// ── UPPER ─────────────────────────────────────────────────────────────────────
rawTorqueUpper := upperMasterTorqueFeedback;
instsFT_PT1UpperTorqueFilter( in := rawTorqueUpper, 
							   T := torqueFilterTime, 
							   K := 1.0, 
							   out => filteredTorqueUpper );
							   

// Master cap and base limit (never exceed master)
capMasterUpper := LIMIT(torqueLimitMinPct, filteredTorqueUpper, torqueLimitMaxPct);
baseLimitUpper := MIN(
    capMasterUpper,
    LIMIT(torqueLimitMinPct, filteredTorqueUpper + slaveTorqueOfsset, torqueLimitMaxPct)
);

IF NOT enableTorquePid THEN
    upperSlave1DriveTorqueRefPct := capMasterUpper;
    upperSlave2DriveTorqueRefPct := capMasterUpper;
ELSE
    directTorqueUpper := LIMIT(torqueLimitMinPct, baseLimitUpper - torqueTrimLimit, capMasterUpper);
    avgTorqueUpper    := 0.5 * (upperSlave1TorqueFeedback + upperSlave2TorqueFeedback);

    instCTRL_PID_UpperTorqueTrim(
        ACT := avgTorqueUpper,
        SET := baseLimitUpper,
        MAN := NOT enableTorquePid,   // manual when disabled (tracks 0)
        M_I := 0.0,
        RST := FALSE,
        KP  := torqueCtrlKp,
        TN  := torqueCtrlTn,
        TV  := torqueCtrlTv,
        LL  := 0.0,                   // unipolar: only add
        LH  := torqueTrimLimit,
        Y   => trimUp
    );

    upperSlave1DriveTorqueRefPct := LIMIT(torqueLimitMinPct, directTorqueUpper + trimUp, capMasterUpper);
    upperSlave2DriveTorqueRefPct := LIMIT(torqueLimitMinPct, directTorqueUpper + trimUp, capMasterUpper);
END_IF;


// ── LOWER ─────────────────────────────────────────────────────────────────────
rawTorqueLower := lowerMasterTorqueFeedback;
instsFT_PT1LowerTorqueFilter( in := rawTorqueLower, T := torqueFilterTime, K := 1.0, out => filteredTorqueLower );

capMasterLower := LIMIT(torqueLimitMinPct, filteredTorqueLower, torqueLimitMaxPct);
baseLimitLower := MIN(
    capMasterLower,
    LIMIT(torqueLimitMinPct, filteredTorqueLower + slaveTorqueOfsset, torqueLimitMaxPct)
);

IF NOT enableTorquePid THEN
    lowerSlave1DriveTorqueRefPct := capMasterLower;
    lowerSlave2DriveTorqueRefPct := capMasterLower;
ELSE
    directTorqueLower := LIMIT(torqueLimitMinPct, baseLimitLower - torqueTrimLimit, capMasterLower);
    avgTorqueLower    := 0.5 * (lowerSlave1TorqueFeedback + lowerSlave2TorqueFeedback);

    instCTRL_PID_LowerTorqueTrim(
        ACT := avgTorqueLower,
        SET := baseLimitLower,
        MAN := NOT enableTorquePid,
        M_I := 0.0,
        RST := FALSE,
        KP  := torqueCtrlKp,
        TN  := torqueCtrlTn,
        TV  := torqueCtrlTv,
        LL  := 0.0,
        LH  := torqueTrimLimit,
        Y   => trimLo
    );

    lowerSlave1DriveTorqueRefPct := LIMIT(torqueLimitMinPct, directTorqueLower + trimLo, capMasterLower);
    lowerSlave2DriveTorqueRefPct := LIMIT(torqueLimitMinPct, directTorqueLower + trimLo, capMasterLower);
END_IF;
END_METHOD

END_FUNCTION_BLOCK

// ---- Function Blocks/PaperMachine/Auxiliary/FB_Gen_SRamp.TcPOU
FUNCTION_BLOCK FB_Gen_SRamp
VAR_INPUT
	X : REAL;
	A_UP : REAL  := 1.0;
	A_DN :REAL  := -1.0;;
	VU_MAX : REAL := 1.0;
	VD_MAX : REAL := -1.0;
	LIMIT_HIGH : REAL := 100.0;
	LIMIT_LOW : REAL := -100.0;
	RST : BOOL;
END_VAR
VAR_OUTPUT
	Y : REAL;
	V : REAL;
END_VAR
VAR
	cycle_time : TC_S;
	init: BOOL;
END_VAR

(* read the system_time in microseconds *)
cycle_time();

(* assure range of inputs *)
A_up := MAX(0.0, A_UP);
A_dn := MIN(0.0, A_dn);
VU_max := MAX(0.0, VU_max);
VD_max := MIN(0.0, VD_MAX);

(* calculate the output offset *)
IF rst OR NOT init THEN
	init := TRUE;
	Y := 0.0;
	V := 0.0;
ELSIF X = Y THEN
	v := 0.0;
ELSIF X > Y THEN
	(* output is too low >> ramp up and brake at the end *)
	(* accelerate the speed and limit to vu_max *)
	v := MIN(v + A_UP * cycle_time.TC, vu_max);
	(* calculate the max speed to be able to brake and select the lowest *)
	v := MIN(SQRT((Y-X) * 2.0 * A_DN), v);
	(* calculate the output and obey limits *)
	y := LIMIT(limit_low, y + MIN(v * cycle_time.TC, X-Y), limit_high);
ELSIF X < Y THEN
	(* output is too high >> ramp dn and brake at the end *)
	(* accelerate the speed and limit to vd_max *)
	v := MAX(v + A_DN * cycle_time.TC, vd_max);
	(* calculate the max speed to be able to brake and select the lowest *)
	v := MAX(-SQRT((Y-X) * 2.0 * A_UP), v);
	(* calculate the output and obey limits *)
	y := LIMIT(limit_low, y + MAX(v * cycle_time.TC, X-Y), limit_high);
END_IF;


(* revision history
hm	13. mar. 2008	rev 1.0
	original version

hm	11. mar. 2009	rev 1.1
	real constants updated to new systax using dot																																																																																																																																																																																																																																																																																																																																																																																																																																																																																																																																																																																																																																																																																																																																																																																																																																																																																																																																																																																																																																																											

*)

END_FUNCTION_BLOCK

// ---- Function Blocks/PaperMachine/DriveControl/FB_PressSectionDriveControl_V2.TcPOU
FUNCTION_BLOCK FB_PressSectionDriveControl_V2

VAR_INPUT

    //────────────────────────────────────────────
    // GROUP / INTERLOCKS
    //────────────────────────────────────────────
    startGroup              : BOOL; // Start command (pulse) / Comando de partida (pulso)
    stopGroup               : BOOL; // Stop command (level) / Comando de parada (nível)
    groupReset              : BOOL; // Fault reset / Reset de falhas do grupo
    groupFastStop           : BOOL;  // EN: Reset group faults / PT: Reset de falhas do grupo
	
    //────────────────────────────────────────────
    // AUXILIARY MOTORS — INDICATORS & COMMANDS
    //────────────────────────────────────────────
    grouSpeedDifIncCmd         : BOOL; // Lamp: offset increasing / Lâmpada: aumento de offset
    grouSpeedDifDecCmd         : BOOL; // Lamp: offset decreasing / Lâmpada: redução de offset
	
    //────────────────────────────────────────────
    // SPEED ADJUSTMENTS / OFFSET TUNING
    //────────────────────────────────────────────
    groupRecoverSpeedCmd    : BOOL; // Recover speed while TRUE / Recuperar velocidade enquanto TRUE


    //────────────────────────────────────────────
    // DRIVE STATUS INPUTS — PRESS SECTION (2 MOTORS)
    //────────────────────────────────────────────
    firstPressReady         : BOOL; // First press (MASTER) ready / Prensa 1 (mestre) pronto
    secondPressReady        : BOOL; // Second press (SLAVE) ready / Prensa 2 (escravo) pronto
	paperPresenceSensor : BOOL;

    //────────────────────────────────────────────
    // SPEED SETPOINTS / MODE
    //────────────────────────────────────────────
    groupAutoSpeedMPM       : REAL; // Auto mode speed [m/min] / Velocidade em modo automático [m/min]
    groupManualSpeedMPM     : REAL := 50.0; // Manual mode speed / Velocidade em modo manual
    groupSpeedAutoMan       : BOOL; // Speed mode: 0=Manual, 1=Auto / Modo de velocidade: 0=Manual, 1=Automático

    //────────────────────────────────────────────
    // SPEED & TORQUE FEEDBACKS
    //────────────────────────────────────────────
    firstPressSpeedFeedback : REAL; // First press speed feedback / Velocidade medida da prensa 1
    firstPressTorqueFeedback: REAL; // First press torque feedback / Torque da prensa 1
    secondPressSpeedFeedback: REAL; // Second press speed feedback / Velocidade medida da prensa 2
    secondPressTorqueFeedback: REAL; // Second press torque feedback / Torque da prensa 2


    //──── Upper Felt 1 Stretcher ────
    upperFelt1StretcherCmdFwd     : BOOL; // Run forward / Comando para frente
    upperFelt1StretcherCmdRev     : BOOL; // Run reverse / Comando para trás
    upperFelt1StretcherFault      : BOOL; // Fault detected / Falha detectada
    upperFelt1StretcherLimitFwd   : BOOL; // End limit forward / Fim de curso frente
    upperFelt1StretcherLimitRev   : BOOL; // End limit reverse / Fim de curso trás

    //──── Upper Felt 2 Stretcher ────
    upperFelt2StretcherCmdFwd     : BOOL; // Run forward / Comando para frente
    upperFeltt2tretcherCmdRev     : BOOL; // Run reverse / Comando para trás (corrigir nome!)
    upperFeltS2tretcherFault      : BOOL; // Fault detected / Falha detectada
    upperFeltS2tretcherLimitFwd   : BOOL; // End limit forward / Fim de curso frente
    upperFeltS2tretcherLimitRev   : BOOL; // End limit reverse / Fim de curso trás

    //──── Lower Felt Stretcher ────
    lowerFeltStretcherCmdFwd      : BOOL;
    lowerFeltStretcherCmdRev      : BOOL;
    lowerFeltStretcherFault       : BOOL;
    lowerFeltStretcherLimitFwd    : BOOL;
    lowerFeltStretcherLimitRev    : BOOL;

    //──── Upper Infeed Roll ────
    upperInfeedRollCmdFwd         : BOOL;
    upperInfeedRollCmdRev         : BOOL;
    upperInfeedRollFault          : BOOL;
    upperInfeedRollLimitFwd       : BOOL;
    upperInfeedRollLimitRev       : BOOL;

    //──── Lower Infeed Roll ────
    lowerInfeedRollCmdFwd         : BOOL;
    lowerInfeedRollCmdRev         : BOOL;
    lowerInfeedRollFault          : BOOL;
    lowerInfeedRollLimitFwd       : BOOL;
    lowerInfeedRollLimitRev       : BOOL;

    //────────────────────────────────────────────
    // FELT EDGE / RUNNING SAFETY SENSORS
    //────────────────────────────────────────────
    pressSectionUpperFelt1OverrunSensorOperatorSide : BOOL; // Operator side / Lado operador
    pressSectionUpperFelt1OverrunSensorDriveSide    : BOOL; // Drive side / Lado comando

    pressSectionUpperFelt2OverrunSensorOperatorSide : BOOL;
    pressSectionUpperFelt2OverrunSensorDriveSide    : BOOL;

    pressSectionLowerFeltOverrunSensorOperatorSide  : BOOL;
    pressSectionLowerFeltOverrunSensorDriveSide     : BOOL;

	
	machineConfig			:  PaperMachine_TypeHmiConfig;
	
END_VAR



VAR_OUTPUT

    //────────────────────────────────────────────
    // STATE / DIAGNOSTICS
    //────────────────────────────────────────────
    deviceState                 : STRING; // Current state string / Estado atual em texto
    statusCode                  : INT;    // 0=Idle, 1=Starting, 2=Running, 3=Fault
    groupFault                  : BOOL;   // TRUE if any group fault active / Falha geral do grupo
	speedDif						: REAL;

    //────────────────────────────────────────────
    // SPEED REFERENCES (TO DRIVES) AND DISPLAY
    //────────────────────────────────────────────
    firstPressSpeedSetpointRPM  		: REAL; // Master speed reference [%] / Referência de velocidade mestre
    secondPressSpeedSetpointRPM 		: REAL; // Slave speed reference [%] / Referência de velocidade escravo 
	
	firstPressSpeedFeedbackRPM  		: REAL; // Master speed reference [%] / Referência de velocidade mestre
    secondPressSpeedFeedbackRPM 		: REAL; // Slave speed reference [%] / Referência de velocidade escravo 
	
	firstPressSpeedFeedbackMPM  		: REAL; // Master speed reference [%] / Referência de velocidade mestre
    secondPressSpeedFeedbackMPM 		: REAL; // Slave speed reference [%] / Referência de velocidade escravo 

	firstPressTorqueFeedbackPct  		: REAL; // Master speed reference [%] / Referência de velocidade mestre
    secondPressTorqueFeedbackPct 		: REAL; // Slave speed reference [%] / Referência de velocidade escravo 
	
	
	nextGroupSpeedRefMPM        : REAL; // Next group speed [m/min] / Velocidade do próximo grupo [m/min]

    //────────────────────────────────────────────
    // TORQUE REFERENCES / LIMITS (SLAVE)
    //────────────────────────────────────────────
    firstPressTorqueRefPct : REAL; // Torque setpoint for slave / Referência de torque escravo
//    secondPressTorqueRefPct : REAL; // Torque setpoint for slave / Referência de torque escravo

    //────────────────────────────────────────────
    // DRIVE COMMANDS (ENABLE / RESET)
    //────────────────────────────────────────────
    firstPressDriveEnable        : BOOL; // Enable master drive / Habilita drive mestre
    firstPressDriveReset         : BOOL; // Reset master drive fault / Reset falha drive mestre
    secondPressDriveEnable       : BOOL; // Enable slave drive / Habilita drive escravo
    secondPressDriveReset        : BOOL; // Reset slave drive fault / Reset falha drive escravo

    //────────────────────────────────────────────
    // STATUS CODES (PER DRIVE)
    //────────────────────────────────────────────
    firstPressStatusCode        : INT; // 0=Idle, 1=Start, 2=Run, 3=Fault / Código de status da prensa 1
    secondPressStatusCode       : INT; // Código de status da prensa 2

    //────────────────────────────────────────────
    // AUXILIARY MOTORS — DIRECT START OUTPUTS
    //────────────────────────────────────────────
    upperFelt1StretcherRunFwd   : BOOL; // Run forward / Rodar para frente
    upperFelt1StretcherRunRev   : BOOL; // Run reverse / Rodar para trás

    upperFelt2StretcherRunFwd   : BOOL;
    upperFelt2StretcherRunRev   : BOOL;

    lowerFeltStretcherRunFwd    : BOOL;
    lowerFeltStretcherRunRev    : BOOL;

    upperInfeedRollRunFwd       : BOOL;
    upperInfeedRollRunRev       : BOOL;

    lowerInfeedRollRunFwd       : BOOL;
    lowerInfeedRollRunRev       : BOOL;

    //────────────────────────────────────────────
    // HMI ALARMS STRUCTURE
    //────────────────────────────────────────────
    hmiAlarms                   : PaperMachine_TypeHmiAlarms; // Alarm structure / Estrutura de alarmes

END_VAR




VAR
 
	instFB_GroupDriveControl_V1 : FB_GroupDriveControl_V1;
	instFB_GroupSpeedControl_V1 : FB_GroupSpeedControl_V1;
	instFB_GroupDisplayFilters_V1 : FB_GroupDisplayFilters_V1;
	instFB_GroupTorqueTrimControl_V1 : FB_GroupTorqueTrimControl_V1;

	instFB_GroupTorqueTrimControl_V2: FB_GroupTorqueTrimControl_V2;
	speedDifError: BOOL;
	speedDifCheck: REAL;
	instTONFeltOverrunDelay: TON;
	instTOF_PaperPresenseDelay: TOF;	
	
END_VAR

VAR PERSISTENT

END_VAR

// ─────────────────────────────────────────────────────────────────────────────
// MAIN CALL SEQUENCE
// ─────────────────────────────────────────────────────────────────────────────

_GroupControl();          // 1) State machine: edges, enables, stop modes
_StateDisplay();
_SpeedDifferenceCheck();  // 4) Speed difference monitor & trip
_auxiliaryControls();

_alarmsDisplay();

METHOD _alarmsDisplay
VAR_INPUT
END_VAR
(*
//==============================================================
// FAULT EVALUATION — PER CONDITION (flags only; no global set)
//==============================================================

//----------------------------
// PRESS SECTION DRIVES
//----------------------------
hmiAlarms.pressSectionFirstPressFaultAlarm  := firstPressVfdFaultFeedback;
hmiAlarms.pressSectionSecondPressFaultAlarm := secondPressVfdFaultFeedback;

//----------------------------
// PRESS SECTION AUXILIARIES
//----------------------------
hmiAlarms.pressSectionUpperFeltStretcherFaultAlarm := upperFelt1StretcherFault;
hmiAlarms.pressSectionLowerFeltStretcherFaultAlarm := lowerFeltStretcherFault;
hmiAlarms.pressSectionUpperInfeedRollFaultAlarm    := upperInfeedRollFault;
hmiAlarms.pressSectionLowerInfeedRollFaultAlarm    := lowerInfeedRollFault;


//==============================================================
// PRESS SECTION — FELT EDGE OVERRUN ALARMS (DIRECT SENSORS)
//==============================================================

hmiAlarms.pressSectionUpperFelt1OverrunOperatorSideAlarm := pressSectionUpperFelt1OverrunSensorOperatorSide;
hmiAlarms.pressSectionUpperFelt1OverrunDriveSideAlarm    := pressSectionUpperFelt1OverrunSensorDriveSide;

hmiAlarms.pressSectionUpperFelt2OverrunOperatorSideAlarm := pressSectionUpperFelt2OverrunSensorOperatorSide;
hmiAlarms.pressSectionUpperFelt2OverrunDriveSideAlarm    := pressSectionUpperFelt2OverrunSensorDriveSide;

hmiAlarms.pressSectionLowerFeltOverrunOperatorSideAlarm := pressSectionLowerFeltOverrunSensorOperatorSide;
hmiAlarms.pressSectionLowerFeltOverrunDriveSideAlarm    := pressSectionLowerFeltOverrunSensorDriveSide;


//----------------------------
// PRESS SECTION GROUP FAULT STATUS
//----------------------------
groupFault :=
    hmiAlarms.pressSectionFirstPressFaultAlarm 
	OR hmiAlarms.pressSectionSecondPressFaultAlarm 
	OR hmiAlarms.pressFelt1OverrunOperatorSideAlarm
	OR hmiAlarms.pressFelt1OverrunDriveSideAlarm
	OR hmiAlarms.pressFelt2OverrunOperatorSideAlarm
	OR hmiAlarms.pressFelt2OverrunDriveSideAlarm
	OR hmiAlarms.pressFelt3OverrunOperatorSideAlarm
	OR hmiAlarms.pressFelt3OverrunDriveSideAlarm;


*)
//==============================================================
// FAULT EVALUATION — PER CONDITION (flags only; no global set)
//==============================================================

//----------------------------
// PRESS SECTION DRIVES
//----------------------------
//hmiAlarms.pressSectionFirstPressFaultAlarm  := firstPressVfdFaultFeedback;
//hmiAlarms.pressSectionSecondPressFaultAlarm := secondPressVfdFaultFeedback;

//----------------------------
// PRESS SECTION AUXILIARIES
//----------------------------
hmiAlarms.pressSectionUpperFeltStretcherFaultAlarm := upperFelt1StretcherFault;
hmiAlarms.pressSectionLowerFeltStretcherFaultAlarm := lowerFeltStretcherFault;
hmiAlarms.pressSectionUpperInfeedRollFaultAlarm    := upperInfeedRollFault;
hmiAlarms.pressSectionLowerInfeedRollFaultAlarm    := lowerInfeedRollFault;


//==============================================================
// PRESS SECTION — FELT EDGE OVERRUN ALARMS (DIRECT SENSORS)
//==============================================================

hmiAlarms.pressSectionUpperFelt1OverrunOperatorSideAlarm := pressSectionUpperFelt1OverrunSensorOperatorSide;
hmiAlarms.pressSectionUpperFelt1OverrunDriveSideAlarm    := pressSectionUpperFelt1OverrunSensorDriveSide;

hmiAlarms.pressSectionUpperFelt2OverrunOperatorSideAlarm := pressSectionUpperFelt2OverrunSensorOperatorSide;
hmiAlarms.pressSectionUpperFelt2OverrunDriveSideAlarm    := pressSectionUpperFelt2OverrunSensorDriveSide;

hmiAlarms.pressSectionLowerFeltOverrunOperatorSideAlarm := pressSectionLowerFeltOverrunSensorOperatorSide;
hmiAlarms.pressSectionLowerFeltOverrunDriveSideAlarm    := pressSectionLowerFeltOverrunSensorDriveSide;


//----------------------------
// PRESS SECTION GROUP FAULT STATUS
//----------------------------
groupFault := hmiAlarms.pressSectionFirstPressFaultAlarm OR
		hmiAlarms.pressSectionSecondPressFaultAlarm OR
		hmiAlarms.pressSectionUpperFelt1OverrunOperatorSideAlarm OR
		hmiAlarms.pressSectionUpperFelt1OverrunDriveSideAlarm OR
		hmiAlarms.pressSectionUpperFelt2OverrunOperatorSideAlarm OR
		hmiAlarms.pressSectionUpperFelt2OverrunDriveSideAlarm OR
		hmiAlarms.pressSectionLowerFeltOverrunOperatorSideAlarm OR
		hmiAlarms.pressSectionLowerFeltOverrunDriveSideAlarm;
END_METHOD

METHOD _auxiliaryControls
VAR_INPUT
END_VAR
//============================
// LOWER FELT STRETCHER
//============================
IF NOT lowerFeltStretcherFault THEN
    IF lowerFeltStretcherCmdFwd AND NOT lowerFeltStretcherCmdRev AND NOT lowerFeltStretcherLimitFwd THEN
        lowerFeltStretcherRunFwd := TRUE;
    ELSE
        lowerFeltStretcherRunFwd := FALSE;
    END_IF;

    IF lowerFeltStretcherCmdRev AND NOT lowerFeltStretcherCmdFwd AND NOT lowerFeltStretcherLimitRev THEN
        lowerFeltStretcherRunRev := TRUE;
    ELSE
        lowerFeltStretcherRunRev := FALSE;
    END_IF;
ELSE
    lowerFeltStretcherRunFwd := FALSE;
    lowerFeltStretcherRunRev := FALSE;
END_IF;


//============================
// UPPER INFEED ROLL
//============================
IF NOT upperInfeedRollFault THEN
    IF upperInfeedRollCmdFwd AND NOT upperInfeedRollCmdRev AND NOT upperInfeedRollLimitFwd THEN
        upperInfeedRollRunFwd := TRUE;
    ELSE
        upperInfeedRollRunFwd := FALSE;
    END_IF;

    IF upperInfeedRollCmdRev AND NOT upperInfeedRollCmdFwd AND NOT upperInfeedRollLimitRev THEN
        upperInfeedRollRunRev := TRUE;
    ELSE
        upperInfeedRollRunRev := FALSE;
    END_IF;
ELSE
    upperInfeedRollRunFwd := FALSE;
    upperInfeedRollRunRev := FALSE;
END_IF;


//============================
// LOWER INFEED ROLL
//============================
IF NOT lowerInfeedRollFault THEN
    IF lowerInfeedRollCmdFwd AND NOT lowerInfeedRollCmdRev AND NOT lowerInfeedRollLimitFwd THEN
        lowerInfeedRollRunFwd := TRUE;
    ELSE
        lowerInfeedRollRunFwd := FALSE;
    END_IF;

    IF lowerInfeedRollCmdRev AND NOT lowerInfeedRollCmdFwd AND NOT lowerInfeedRollLimitRev THEN
        lowerInfeedRollRunRev := TRUE;
    ELSE
        lowerInfeedRollRunRev := FALSE;
    END_IF;
ELSE
    lowerInfeedRollRunFwd := FALSE;
    lowerInfeedRollRunRev := FALSE;
END_IF;


//============================
// UPPER FELT 1 STRETCHER
//============================
IF NOT upperFelt1StretcherFault THEN
    IF upperFelt1StretcherCmdFwd AND NOT upperFelt1StretcherCmdRev AND NOT upperFelt1StretcherLimitFwd THEN
        upperFelt1StretcherRunFwd := TRUE;
    ELSE
        upperFelt1StretcherRunFwd := FALSE;
    END_IF;

    IF upperFelt1StretcherCmdRev AND NOT upperFelt1StretcherCmdFwd AND NOT upperFelt1StretcherLimitRev THEN
        upperFelt1StretcherRunRev := TRUE;
    ELSE
        upperFelt1StretcherRunRev := FALSE;
    END_IF;
ELSE
    upperFelt1StretcherRunFwd := FALSE;
    upperFelt1StretcherRunRev := FALSE;
END_IF;

//============================
// UPPER FELT 2 STRETCHER
//============================
IF NOT upperFeltS2tretcherFault THEN
    IF upperFelt2StretcherCmdFwd AND NOT upperFeltt2tretcherCmdRev AND NOT upperFeltS2tretcherLimitFwd THEN
        upperFelt2StretcherRunFwd := TRUE;
    ELSE
        upperFelt2StretcherRunFwd := FALSE;
    END_IF;

    IF upperFeltt2tretcherCmdRev AND NOT upperFelt2StretcherCmdFwd AND NOT upperFeltS2tretcherLimitRev THEN
        upperFelt2StretcherRunRev := TRUE;
    ELSE
        upperFelt2StretcherRunRev := FALSE;
    END_IF;
ELSE
    upperFelt2StretcherRunFwd := FALSE;
    upperFelt2StretcherRunRev := FALSE;
END_IF;
END_METHOD

METHOD _GroupControl
VAR_INPUT
END_VAR
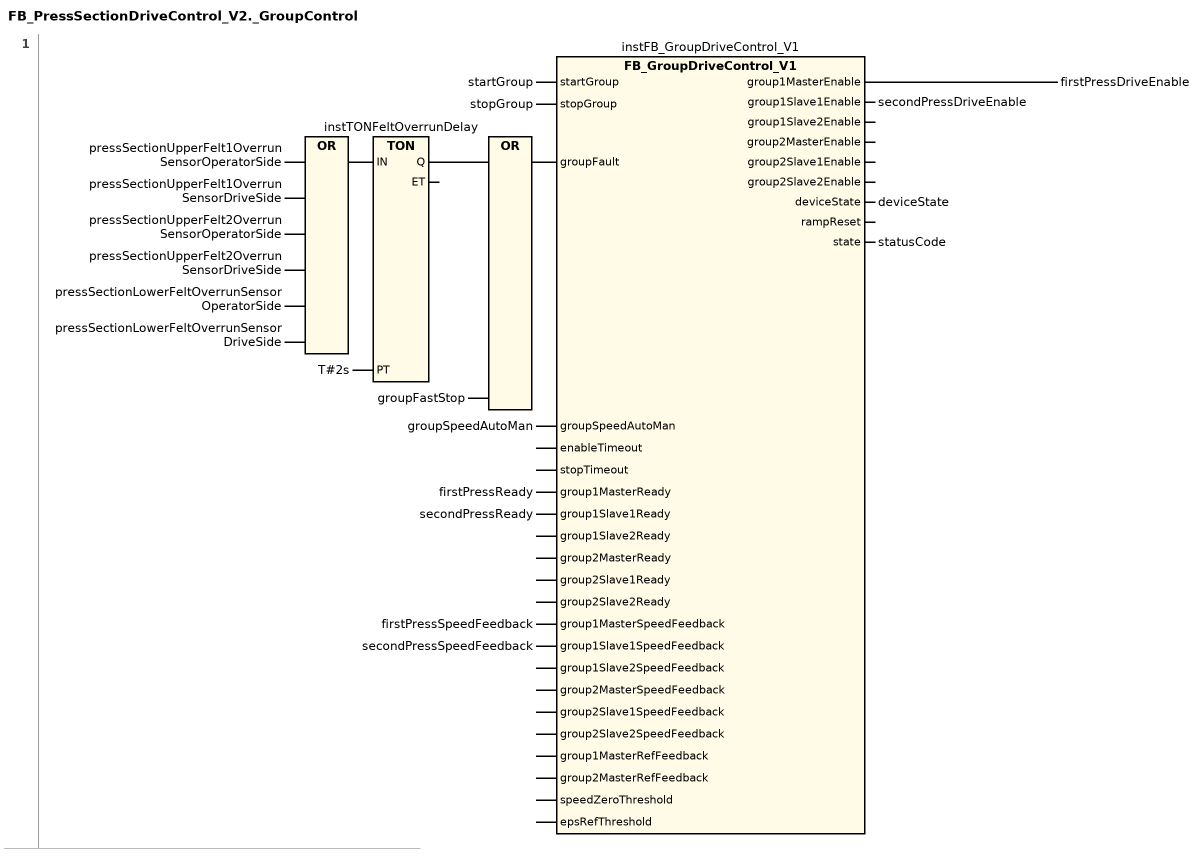
// NETWORK 1
instTONFeltOverrunDelay(IN := pressSectionUpperFelt1OverrunSensorOperatorSide OR pressSectionUpperFelt1OverrunSensorDriveSide OR pressSectionUpperFelt2OverrunSensorOperatorSide OR pressSectionUpperFelt2OverrunSensorDriveSide OR pressSectionLowerFeltOverrunSensorOperatorSide OR pressSectionLowerFeltOverrunSensorDriveSide, PT := T#2s); // TON
instFB_GroupDriveControl_V1(
    startGroup := startGroup,
    stopGroup := stopGroup,
    groupFault := instTONFeltOverrunDelay.Q OR groupFastStop,
    groupSpeedAutoMan := groupSpeedAutoMan,
    group1MasterReady := firstPressReady,
    group1Slave1Ready := secondPressReady,
    group1MasterSpeedFeedback := firstPressSpeedFeedback,
    group1Slave1SpeedFeedback := secondPressSpeedFeedback,
    group1Slave1Enable => secondPressDriveEnable,
    deviceState => deviceState,
    state => statusCode); // FB_GroupDriveControl_V1
firstPressDriveEnable := instFB_GroupDriveControl_V1.group1MasterEnable;

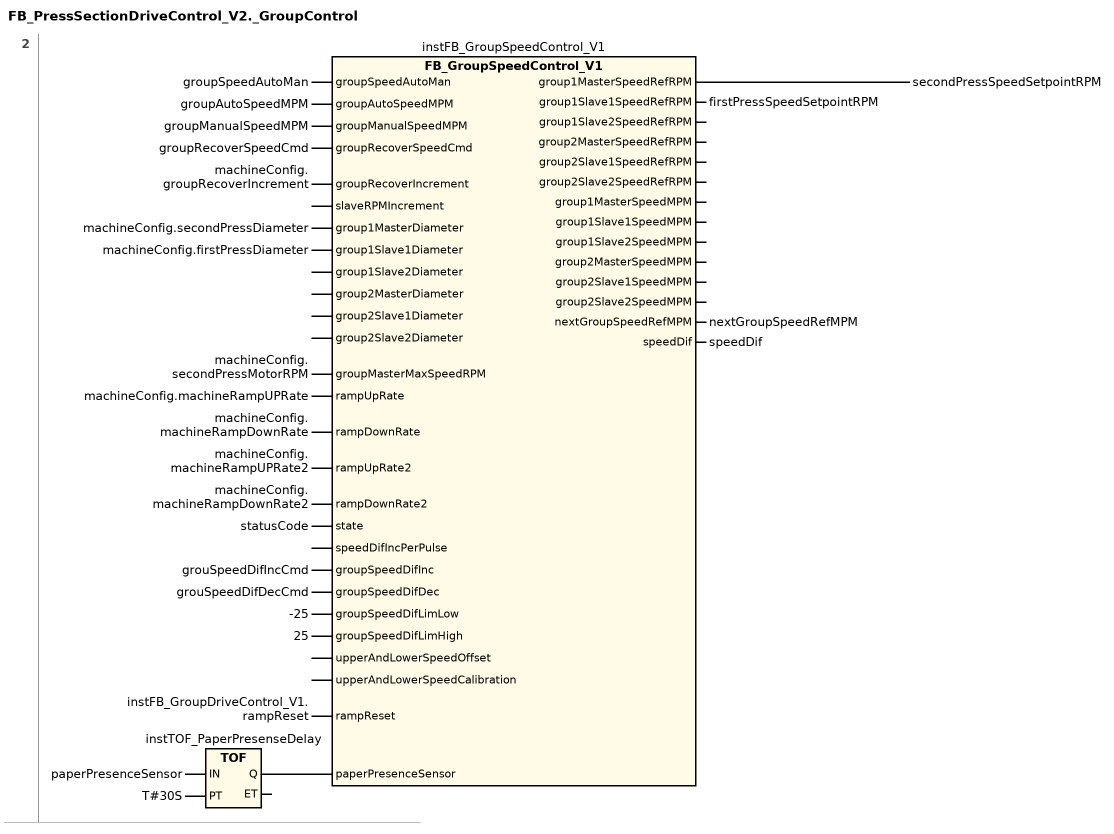
// NETWORK 2
instTOF_PaperPresenseDelay(IN := paperPresenceSensor, PT := T#30S); // TOF
instFB_GroupSpeedControl_V1(
    groupSpeedAutoMan := groupSpeedAutoMan,
    groupAutoSpeedMPM := groupAutoSpeedMPM,
    groupManualSpeedMPM := groupManualSpeedMPM,
    groupRecoverSpeedCmd := groupRecoverSpeedCmd,
    groupRecoverIncrement := machineConfig.groupRecoverIncrement,
    group1MasterDiameter := machineConfig.secondPressDiameter,
    group1Slave1Diameter := machineConfig.firstPressDiameter,
    groupMasterMaxSpeedRPM := machineConfig.secondPressMotorRPM,
    rampUpRate := machineConfig.machineRampUPRate,
    rampDownRate := machineConfig.machineRampDownRate,
    rampUpRate2 := machineConfig.machineRampUPRate2,
    rampDownRate2 := machineConfig.machineRampDownRate2,
    state := statusCode,
    groupSpeedDifInc := grouSpeedDifIncCmd,
    groupSpeedDifDec := grouSpeedDifDecCmd,
    groupSpeedDifLimLow := -25,
    groupSpeedDifLimHigh := 25,
    rampReset := instFB_GroupDriveControl_V1.rampReset,
    paperPresenceSensor := instTOF_PaperPresenseDelay.Q,
    group1Slave1SpeedRefRPM => firstPressSpeedSetpointRPM,
    nextGroupSpeedRefMPM => nextGroupSpeedRefMPM,
    speedDif => speedDif); // FB_GroupSpeedControl_V1
secondPressSpeedSetpointRPM := instFB_GroupSpeedControl_V1.group1MasterSpeedRefRPM;

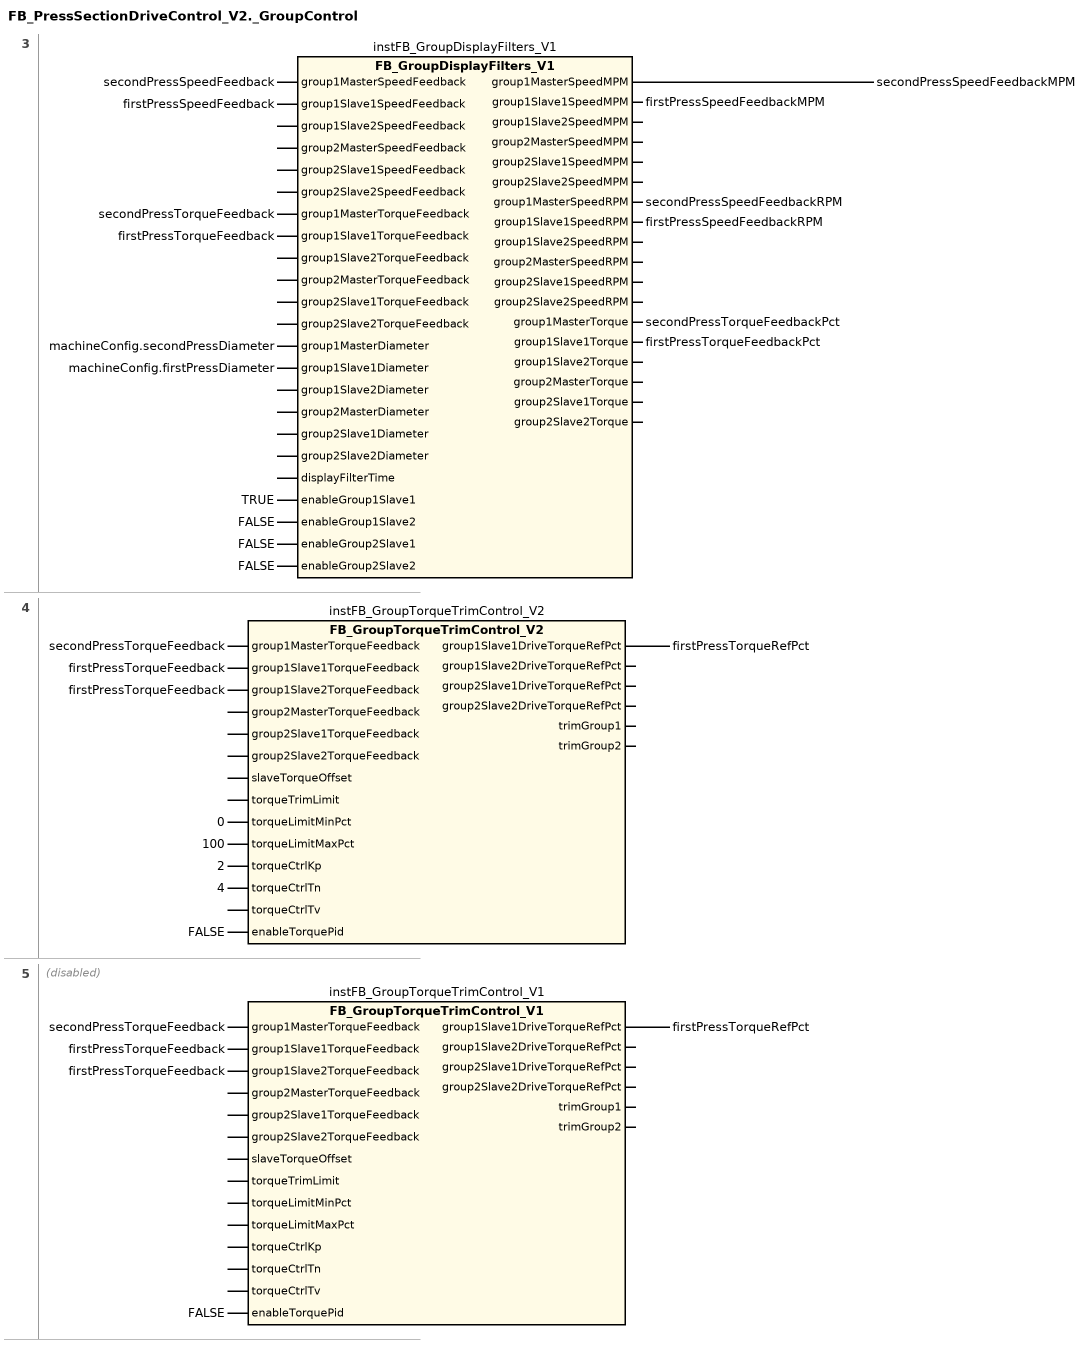
// NETWORK 3
instFB_GroupDisplayFilters_V1(
    group1MasterSpeedFeedback := secondPressSpeedFeedback,
    group1Slave1SpeedFeedback := firstPressSpeedFeedback,
    group1MasterTorqueFeedback := secondPressTorqueFeedback,
    group1Slave1TorqueFeedback := firstPressTorqueFeedback,
    group1MasterDiameter := machineConfig.secondPressDiameter,
    group1Slave1Diameter := machineConfig.firstPressDiameter,
    enableGroup1Slave1 := TRUE,
    enableGroup1Slave2 := FALSE,
    enableGroup2Slave1 := FALSE,
    enableGroup2Slave2 := FALSE,
    group1Slave1SpeedMPM => firstPressSpeedFeedbackMPM,
    group1MasterSpeedRPM => secondPressSpeedFeedbackRPM,
    group1Slave1SpeedRPM => firstPressSpeedFeedbackRPM,
    group1MasterTorque => secondPressTorqueFeedbackPct,
    group1Slave1Torque => firstPressTorqueFeedbackPct); // FB_GroupDisplayFilters_V1
secondPressSpeedFeedbackMPM := instFB_GroupDisplayFilters_V1.group1MasterSpeedMPM;

// NETWORK 4
instFB_GroupTorqueTrimControl_V2(
    group1MasterTorqueFeedback := secondPressTorqueFeedback,
    group1Slave1TorqueFeedback := firstPressTorqueFeedback,
    group1Slave2TorqueFeedback := firstPressTorqueFeedback,
    torqueLimitMinPct := 0,
    torqueLimitMaxPct := 100,
    torqueCtrlKp := 2,
    torqueCtrlTn := 4,
    enableTorquePid := FALSE); // FB_GroupTorqueTrimControl_V2
firstPressTorqueRefPct := instFB_GroupTorqueTrimControl_V2.group1Slave1DriveTorqueRefPct;

// NETWORK 5 (disabled)
// instFB_GroupTorqueTrimControl_V1(
//     group1MasterTorqueFeedback := secondPressTorqueFeedback,
//     group1Slave1TorqueFeedback := firstPressTorqueFeedback,
//     group1Slave2TorqueFeedback := firstPressTorqueFeedback,
//     enableTorquePid := FALSE); // FB_GroupTorqueTrimControl_V1
// firstPressTorqueRefPct := instFB_GroupTorqueTrimControl_V1.group1Slave1DriveTorqueRefPct;
END_METHOD

METHOD PRIVATE _Scale : REAL
VAR_INPUT
    X    : REAL;
    I_LO : REAL;
    I_HI : REAL;
    O_LO : REAL;
    O_HI : REAL;
END_VAR
IF I_LO = I_HI THEN
	_Scale := O_LO;
ELSE
	_Scale := (O_HI - O_LO) / (I_HI - I_LO) * (LIMIT(I_LO, X, I_HI) - I_LO) + O_LO;
END_IF;
END_METHOD

// ============================== Methods ==============================
// Intra-section speed supervision for Press Section (firstPress ↔ secondPress)
METHOD _SpeedDifferenceCheck
VAR_INPUT
END_VAR
VAR
    diffPress : REAL;   // Absolute speed difference between master and slave
END_VAR

(*
    //────────────────────────────────────────────
    firstPressSpeedFeedback : REAL; // First press speed feedback / Velocidade medida da prensa 1
    firstPressTorqueFeedback: REAL; // First press torque feedback / Torque da prensa 1
    secondPressSpeedFeedback: REAL; // Second press speed feedback / Velocidade medida da prensa 2
    secondPressTorqueFeedback: REAL; // Second press torque feedback / Torque da prensa 2

*)


speedDifCheck := ABS(secondPressSpeedFeedbackMPM - firstPressSpeedFeedbackMPM);


IF speedDifCheck > 10 THEN
	
	speedDifError := TRUE;
	
	ELSE
		
	speedDifError := FALSE;
	
	
END_IF
END_METHOD

METHOD _StateDisplay
VAR_INPUT
END_VAR

// ──────────────────────────────────────────────────────────────────────────────
// _StateDisplay — Press Section (firstPress = Master, secondPress = Slave)
// Maps the internal machine "state" to a compact HMI status code and derives
// per-drive motor status codes from VFD signals.
//
// statusCode / firstPressStatusCode / secondPressStatusCode legend:
//   0 = Idle, 1 = Starting, 2 = Running, 3 = Fault
//
// Machine "state" groups:
//   0 = IDLE, 1 = ENABLE, 2 = WAIT_EN, 3 = RAMP_EN, 4 = RUN, 5 = STOPPING, 10 = FAULT
// Priority rule (for motors): Fault > Running > Starting > Idle
// ──────────────────────────────────────────────────────────────────────────────
VAR CONSTANT
    STATUS_IDLE     : INT := 0;
    STATUS_STARTING : INT := 1;
    STATUS_RUNNING  : INT := 2;
    STATUS_FAULT    : INT := 3;
END_VAR
(*
// ─────────────── Group machine states into a single HMI statusCode ───────────
CASE state OF
    10: // FAULT
        statusCode := STATUS_FAULT;
    4:  // RUN
        statusCode := STATUS_RUNNING;
    1, 2, 3: // ENABLE / WAIT_EN / RAMP_EN
        statusCode := STATUS_STARTING;
ELSE   // IDLE, STOPPING, or any other
        statusCode := STATUS_IDLE;
END_CASE;


// ─────────────── Per-drive status (priority: Fault > Running > Starting > Idle) ───────────────
// FIRST PRESS (MASTER)
IF firstPressVfdFaultFeedback THEN
    firstPressStatusCode := STATUS_FAULT;
ELSIF firstPressVfdRunFeedback THEN
    firstPressStatusCode := STATUS_RUNNING;
ELSIF firstPressDriveEnable THEN
    firstPressStatusCode := STATUS_STARTING;
ELSE
    firstPressStatusCode := STATUS_IDLE;
END_IF;

// SECOND PRESS (SLAVE)
IF secondPressVfdFaultFeedback THEN
    secondPressStatusCode := STATUS_FAULT;
ELSIF secondPressVfdRunFeedback THEN
    secondPressStatusCode := STATUS_RUNNING;
ELSIF secondPressDriveEnable THEN
    secondPressStatusCode := STATUS_STARTING;
ELSE
    secondPressStatusCode := STATUS_IDLE;
END_IF;
*)
END_METHOD

END_FUNCTION_BLOCK

// ---- Function Blocks/PaperMachine/FB_GroupDriveControl_V1.TcPOU
FUNCTION_BLOCK FB_GroupDriveControl_V1
VAR_INPUT
    //----------------------------------------------------------------------
    // GROUP COMMANDS
    //----------------------------------------------------------------------
    startGroup              : BOOL;      // EN: Start command (pulse) / PT: Comando de partida (pulso)
    stopGroup               : BOOL;      // EN: Stop command (maintained) / PT: Comando de parada (mantido)
    groupFault              : BOOL;      // EN: External fault signal / PT: Falha externa do grupo
    groupSpeedAutoMan       : BOOL;      // EN: Mode selector (TRUE=Auto / FALSE=Manual)
    enableTimeout           : TIME := T#5s;   // EN: Timeout for enable feedback / PT: Tempo máx. para habilitação
    stopTimeout             : TIME := T#10s;  // EN: Timeout for controlled stop / PT: Tempo máx. para parada

    //----------------------------------------------------------------------
    // DRIVE STATUS FEEDBACKS
    //----------------------------------------------------------------------
    group1MasterReady       : BOOL := TRUE;  
    group1Slave1Ready       : BOOL := TRUE;  
    group1Slave2Ready       : BOOL := TRUE;  
    group2MasterReady       : BOOL := TRUE;  
    group2Slave1Ready       : BOOL := TRUE;  
    group2Slave2Ready       : BOOL := TRUE;  

    //----------------------------------------------------------------------
    // SPEED FEEDBACKS (RPM or %)
    //----------------------------------------------------------------------
    group1MasterSpeedFeedback : REAL;
    group1Slave1SpeedFeedback : REAL;
    group1Slave2SpeedFeedback : REAL;
    group2MasterSpeedFeedback : REAL;
    group2Slave1SpeedFeedback : REAL;
    group2Slave2SpeedFeedback : REAL;

    //----------------------------------------------------------------------
    // DRIVE REFERENCE FEEDBACKS (for zero check)
    //----------------------------------------------------------------------
    group1MasterRefFeedback  : REAL;
    group2MasterRefFeedback  : REAL;

    //----------------------------------------------------------------------
    // THRESHOLDS
    //----------------------------------------------------------------------
    speedZeroThreshold       : REAL := 1.0;   // EN: Threshold to consider stopped / PT: Limite para considerar parado
    epsRefThreshold          : REAL := 1.0;   // EN: Threshold for null reference / PT: Limite de referência nula
END_VAR


VAR_OUTPUT
    //----------------------------------------------------------------------
    // DRIVE ENABLE OUTPUTS
    //----------------------------------------------------------------------
    group1MasterEnable       : BOOL;
    group1Slave1Enable       : BOOL;
    group1Slave2Enable       : BOOL;
    group2MasterEnable       : BOOL;
    group2Slave1Enable       : BOOL;
    group2Slave2Enable       : BOOL;

    //----------------------------------------------------------------------
    // STATUS OUTPUTS
    //----------------------------------------------------------------------
    deviceState              : STRING;   // EN: Current textual state / PT: Estado atual em texto
    rampReset                : BOOL;     // EN: Ramp reset output / PT: Saída de reset da rampa
    state                    : INT;      // EN: Internal state / PT: Estado interno
END_VAR


VAR
    //----------------------------------------------------------------------
    // INTERNAL FLAGS AND TIMERS
    //----------------------------------------------------------------------
    rStart, rStop            : BOOL;
    startGroupOld, stopGroupOld : BOOL;

    allReady, anyFault       : BOOL;
    speedsNearZero, refsNearZero : BOOL;

    instTONEnableWait        : TON;
    instTONStopWait          : TON;
END_VAR

//────────────────────────────────────────────────────────────
// 1) Edge detection for start/stop commands
//────────────────────────────────────────────────────────────
rStart := startGroup AND NOT startGroupOld;   // Rising edge → Start
rStop  := stopGroup  AND NOT stopGroupOld;    // Rising edge → Stop
startGroupOld := startGroup;
stopGroupOld  := stopGroup;

//────────────────────────────────────────────────────────────
// 2) Group readiness and fault aggregation
//────────────────────────────────────────────────────────────
// EN: allReady = all drives are ready
//     anyFault = any drive NOT ready OR external group fault
// PT: allReady = todos os inversores prontos
//     anyFault = algum inversor não pronto OU falha externa
//────────────────────────────────────────────────────────────
allReady :=
    group1MasterReady AND group1Slave1Ready AND group1Slave2Ready AND
    group2MasterReady AND group2Slave1Ready AND group2Slave2Ready;

anyFault :=
    groupFault OR
    NOT group1MasterReady OR NOT group1Slave1Ready OR NOT group1Slave2Ready OR
    NOT group2MasterReady OR NOT group2Slave1Ready OR NOT group2Slave2Ready;

//────────────────────────────────────────────────────────────
// 3) Speed and reference near-zero detection
//────────────────────────────────────────────────────────────
speedsNearZero :=
    (ABS(group1MasterSpeedFeedback) <= speedZeroThreshold) AND
    (ABS(group1Slave1SpeedFeedback) <= speedZeroThreshold) AND
    (ABS(group1Slave2SpeedFeedback) <= speedZeroThreshold) AND
    (ABS(group2MasterSpeedFeedback) <= speedZeroThreshold) AND
    (ABS(group2Slave1SpeedFeedback) <= speedZeroThreshold) AND
    (ABS(group2Slave2SpeedFeedback) <= speedZeroThreshold);

refsNearZero :=
    (ABS(group1MasterRefFeedback) <= epsRefThreshold) AND
    (ABS(group2MasterRefFeedback) <= epsRefThreshold);

//────────────────────────────────────────────────────────────
// 4) State machine — generic dual-group drive controller
//────────────────────────────────────────────────────────────
CASE state OF

    //------------------------------------------------------------------
    0: // IDLE
    //------------------------------------------------------------------
        deviceState := 'IDLE';
        rampReset   := TRUE;

        group1MasterEnable := FALSE;
        group1Slave1Enable := FALSE;
        group1Slave2Enable := FALSE;
        group2MasterEnable := FALSE;
        group2Slave1Enable := FALSE;
        group2Slave2Enable := FALSE;

        IF rStart AND NOT anyFault THEN
            state := 1;
        END_IF

    //------------------------------------------------------------------
    1: // ENABLE_DRIVES
    //------------------------------------------------------------------
        deviceState := 'ENABLE_DRIVES';
        rampReset   := TRUE;

        group1MasterEnable := TRUE;
        group1Slave1Enable := TRUE;
        group1Slave2Enable := TRUE;
        group2MasterEnable := TRUE;
        group2Slave1Enable := TRUE;
        group2Slave2Enable := TRUE;

        instTONEnableWait(IN := TRUE, PT := enableTimeout);

        IF rStop OR stopGroup THEN
            instTONEnableWait(IN := FALSE);
            state := 5;
        ELSE
            state := 2;
        END_IF

    //------------------------------------------------------------------
    2: // WAIT_ENABLE_FEEDBACK
    //------------------------------------------------------------------
        deviceState := 'WAIT_ENABLE_FEEDBACK';
        rampReset   := TRUE;

        instTONEnableWait(IN := TRUE, PT := enableTimeout);

        IF anyFault THEN
            instTONEnableWait(IN := FALSE);
            state := 10; // FAULT
        ELSIF rStop OR stopGroup THEN
            instTONEnableWait(IN := FALSE);
            state := 5;  // STOPPING
        ELSIF allReady THEN
            instTONEnableWait(IN := FALSE);
            state := 3;  // RAMP_ENABLE
        ELSIF instTONEnableWait.Q THEN
            instTONEnableWait(IN := FALSE);
            state := 10; // Timeout fault
        END_IF

    //------------------------------------------------------------------
    3: // RAMP_ENABLE
    //------------------------------------------------------------------
        deviceState := 'RAMP_ENABLE';
        rampReset   := FALSE; // release ramp

        IF rStop OR stopGroup THEN
            state := 5;
        ELSE
            state := 4; // RUN
        END_IF

    //------------------------------------------------------------------
    4: // RUN
    //------------------------------------------------------------------
        deviceState := SEL(groupSpeedAutoMan, 'RUN (Manual)', 'RUN (Auto)');
        rampReset   := FALSE;

        IF anyFault THEN
            state := 10;
        ELSIF rStop OR stopGroup THEN
            state := 5;
        END_IF

    //------------------------------------------------------------------
    5: // STOPPING (controlled deceleration)
    //------------------------------------------------------------------
        deviceState := 'STOPPING';
        rampReset   := FALSE;

        IF anyFault THEN
            state := 10;
        ELSIF speedsNearZero AND refsNearZero THEN
            // Stop complete → disable drives
            group1MasterEnable := FALSE;
            group1Slave1Enable := FALSE;
            group1Slave2Enable := FALSE;
            group2MasterEnable := FALSE;
            group2Slave1Enable := FALSE;
            group2Slave2Enable := FALSE;
            state := 0; // IDLE
        END_IF

    //------------------------------------------------------------------
    10: // FAULT
    //------------------------------------------------------------------
        deviceState := 'FAULT';
        rampReset   := TRUE;

        group1MasterEnable := FALSE;
        group1Slave1Enable := FALSE;
        group1Slave2Enable := FALSE;
        group2MasterEnable := FALSE;
        group2Slave1Enable := FALSE;
        group2Slave2Enable := FALSE;

        // Return to IDLE when faults clear and start released
        IF (NOT anyFault) AND (NOT startGroup) THEN
            state := 0;
        END_IF
END_CASE

END_FUNCTION_BLOCK

// ---- Function Blocks/PaperMachine/FB_GroupTorqueTrimControl_V2.TcPOU
FUNCTION_BLOCK FB_GroupTorqueTrimControl_V2
VAR_INPUT
    //----------------------------------------------------------------------
    // TORQUE FEEDBACKS (already filtered)
    //----------------------------------------------------------------------
    group1MasterTorqueFeedback     : REAL;  // EN: Master torque feedback [% or Nm]
    group1Slave1TorqueFeedback     : REAL;  // EN: Slave 1 torque feedback [% or Nm]
    group1Slave2TorqueFeedback     : REAL;  // EN: Slave 2 torque feedback [% or Nm]
    group2MasterTorqueFeedback     : REAL;  // EN: Master torque feedback [% or Nm]
    group2Slave1TorqueFeedback     : REAL;  // EN: Slave 1 torque feedback [% or Nm]
    group2Slave2TorqueFeedback     : REAL;  // EN: Slave 2 torque feedback [% or Nm]

    //----------------------------------------------------------------------
    // CONFIGURATION PARAMETERS
    //----------------------------------------------------------------------
    slaveTorqueOffset              : REAL := 0.0;     // EN: Fixed offset between master and slave [%]
    torqueTrimLimit                : REAL := 10.0;    // EN: Max PID trim output [%]
    torqueLimitMinPct              : REAL := -10.0;     // EN: Min torque command limit [%]
    torqueLimitMaxPct              : REAL := 10.0;   // EN: Max torque command limit [%]

	
	upperAndLowerDifMinPct :  REAL :=  0.1;
	upperAndLowerDifMaxPct	: REAL := -0.1;
	   
	
    //----------------------------------------------------------------------
    // PID GAINS
    //----------------------------------------------------------------------
    torqueCtrlKp                   : REAL := 1.0;
    torqueCtrlTn                   : REAL := 8.0;
    torqueCtrlTv                   : REAL := 0.0;

    upperAndLowerPIDCtrlKp                   : REAL := 0.10;
    upperAndLowerPIDCtrlTn                   : REAL := 1.0;
    tupperAndLowerPIDCtrlTv                   : REAL := 0.0;
	
	
	enableUpperLowerSpeedTrim			: BOOL;
	
    //----------------------------------------------------------------------
    // CONTROL FLAGS
    //----------------------------------------------------------------------
    enableTorquePid                : BOOL := TRUE;    // EN: Enables PID control (FALSE = fixed torque)
END_VAR


VAR_OUTPUT
    //----------------------------------------------------------------------
    // TORQUE REFERENCES (%)
    //----------------------------------------------------------------------
    group1Slave1DriveTorqueRefPct  : REAL;
    group1Slave2DriveTorqueRefPct  : REAL;
    group2Slave1DriveTorqueRefPct  : REAL;
    group2Slave2DriveTorqueRefPct  : REAL;

    //----------------------------------------------------------------------
    // INTERNAL PID OUTPUTS (for monitoring)
    //----------------------------------------------------------------------
    trimGroup1                     : REAL;
    trimGroup2                     : REAL;
	
	
	upperAndLowerSpeedTrim	 	: REAL;
	
	
END_VAR


VAR
    //----------------------------------------------------------------------
    // INTERNAL PID CONTROLLERS
    //----------------------------------------------------------------------
    instCTRL_PID_Group1TorqueTrim  : CTRL_PID;
    instCTRL_PID_Group2TorqueTrim  : CTRL_PID;
    instCTRL_PID_UpperAndLowerSpdTrim  : CTRL_PID;

	
    //----------------------------------------------------------------------
    // INTERNAL SIGNALS
    //----------------------------------------------------------------------
    capMasterGroup1                : REAL;
    capMasterGroup2                : REAL;
    baseLimitGroup1                : REAL;
    baseLimitGroup2                : REAL;
    directTorqueGroup1             : REAL;
    directTorqueGroup2             : REAL;
    avgTorqueGroup1                : REAL;
    avgTorqueGroup2                : REAL;
	upperAndLowerTorqueDif: REAL;
END_VAR


    instCTRL_PID_Group1TorqueTrim(
        ACT := group1Slave1TorqueFeedback,
        SET := group1MasterTorqueFeedback - slaveTorqueOffset,
        MAN := FALSE,
        M_I := 0.0,
        RST := FALSE,
        KP  := torqueCtrlKp,
        TN  := torqueCtrlTn,
        TV  := torqueCtrlTv,
        LL  := torqueLimitMinPct,                   // Bipolar output
        LH  := torqueLimitMaxPct,
		SUP := 1,
        Y   => group1Slave1DriveTorqueRefPct
    );


	
    instCTRL_PID_Group2TorqueTrim(
        ACT := group2Slave1TorqueFeedback,
        SET := group2MasterTorqueFeedback,
        MAN := FALSE,
        M_I := 0.0,
        RST := FALSE,
        KP  := torqueCtrlKp,
        TN  := torqueCtrlTn,
        TV  := torqueCtrlTv,
        LL  := torqueLimitMinPct,                   // Bipolar output
        LH  := torqueLimitMaxPct,
		SUP := 1,		
        Y   => group2Slave1DriveTorqueRefPct
    );


	IF enableUpperLowerSpeedTrim THEN
		
		instCTRL_PID_UpperAndLowerSpdTrim.LL := upperAndLowerDifMinPct;
		instCTRL_PID_UpperAndLowerSpdTrim.LH := upperAndLowerDifMaxPct;
	
	
	ELSE
		
		instCTRL_PID_UpperAndLowerSpdTrim.LL := 0.0;
		instCTRL_PID_UpperAndLowerSpdTrim.LH := 0.0;	
	
	END_IF
	
	
	
		upperAndLowerTorqueDif := group1MasterTorqueFeedback - group2MasterTorqueFeedback;
	
	    instCTRL_PID_UpperAndLowerSpdTrim(
        ACT := upperAndLowerTorqueDif,
        SET := 0,
        MAN := FALSE,
        M_I := 0.0,
        RST := FALSE,
		SUP := 1,
        KP  := upperAndLowerPIDCtrlKp,
        TN  := upperAndLowerPIDCtrlTn,
        TV  := tupperAndLowerPIDCtrlTv,
//        LL  := upperAndLowerDifMinPct,                   // Bipolar output
//        LH  := upperAndLowerDifMaxPct,
        Y   => upperAndLowerSpeedTrim
    );

END_FUNCTION_BLOCK

// ---- Function Blocks/PaperMachine/Auxiliary/FB_PressureControl.TcPOU
FUNCTION_BLOCK FB_PressureControl
VAR_INPUT
    // Sequence commands
    startCommand            : BOOL;  // Start command (Comando de partida)
    stopCommand             : BOOL;  // Stop command  (Comando de parada)

    // Mode
    autoMode                : BOOL;  // TRUE=Automatic / FALSE=Manual (TRUE=Automático / FALSE=Manual)

    // Process signals (engineering units for pressure)
    pressureFeedback        : REAL;  // Process feedback (Pressão medida)
    autoSetpoint            : REAL;  // Auto mode setpoint (Setpoint de pressão no modo automático)

    // Manual output (direct % command to final element)
    manualOutputPct         : REAL;  // 0..100% manual output (Saída manual 0..100%)

    // PID parameters (OSCAT CTRL_PID) — initial conservative tuning
    kp                      : REAL := 0.8;   // Proportional gain (Ganho proporcional)
    tn                      : REAL := 3.0;   // Integral time [s] (Tempo integral)
    tv                      : REAL := 0.0;   // Derivative time [s] (Tempo derivativo)

    // Output limits and adjustments
    outLowLimitPct          : REAL := 0.0;    // Lower output limit % (Limite inferior da saída)
    outHighLimitPct         : REAL := 100.0;  // Upper output limit % (Limite superior da saída)
    outputOffsetPct         : REAL := 0.0;    // Output offset % (Offset da saída)

    // PID control housekeeping
    resetPID                : BOOL;  // Reset integrator (Zerar integrador)

    // ===== Input filter controls (OSCAT PT1) =====
    enableInputFilter       : BOOL;        // TRUE=apply PT1, FALSE=bypass (Habilita filtro PT1)
    inputFilterTime         : TIME := T#300ms; // PT1 time constant (Constante de tempo)
    inputFilterGainK        : REAL := 1.0; // PT1 gain (Ganho do PT1, tipicamente 1.0)
END_VAR

VAR_OUTPUT
    running                 : BOOL;  // TRUE while in RUN state (TRUE enquanto em operação)
    controlOutputPct        : REAL;  // Final control output 0..100% (Saída final 0..100%)
    pidDiff                 : REAL;  // PID difference (Diferença PID)
    pidLimited              : BOOL;  // TRUE if PID is at limit (TRUE se PID saturado)
END_VAR

VAR
    // State machine
    step                    : INT;   // 0=Idle, 10=Starting, 20=Running, 90=Stopping
    startOld                : BOOL;
    rStart                  : BOOL;

    // Internal / helpers
    manualCmd               : REAL;
    yPID                    : REAL;

    // Filtered feedback
    pressureFeedbackFiltered: REAL;

    // OSCAT instances
    instPID                 : CTRL_PID;
    instsFT_PT1TInputFilter : FT_PT1;   // PT1 filter instance
END_VAR


// ============================ Edges ============================
rStart := startCommand AND NOT startOld;
startOld := startCommand;

// ============================ Stop handling =====================
IF stopCommand THEN
    controlOutputPct := 0.0;
    running := FALSE;
    step := 0;
END_IF


// ============================ State machine =====================
CASE step OF
    // ------------------------------------------------------------
    0: // Idle (Repouso)
        running := FALSE;
        controlOutputPct := 0.0;

        IF rStart AND NOT stopCommand THEN
            step := 10;   // go to starting
        END_IF

    // ------------------------------------------------------------
    10: // Starting (Partida)
        running := TRUE;
        step := 20;

    // ------------------------------------------------------------
    20: // Running (Operando)
        running := TRUE;

        // --- Input filtering (PT1) ---
        _InputFilter(
            enableFilter  := enableInputFilter,
            rawValue      := pressureFeedback,
            filterTime    := inputFilterTime,
            filterGainK   := inputFilterGainK,
            filteredValue => pressureFeedbackFiltered
        );

        // 1) Bound manual command to 0..100%
        manualCmd := manualOutputPct;
        IF manualCmd < 0.0 THEN manualCmd := 0.0; END_IF;
        IF manualCmd > 100.0 THEN manualCmd := 100.0; END_IF;

        // 2) Call OSCAT PID (with bumpless transfer)
        instPID(
            ACT := pressureFeedbackFiltered,  // use filtered feedback
            SET := autoSetpoint,
            M_I := manualCmd,
            MAN := NOT autoMode,
            RST := resetPID,
            KP  := kp,
            TN  := tn,
            TV  := tv,
            LL  := outLowLimitPct,
            LH  := outHighLimitPct,
            Y   => yPID,
            DIFF=> pidDiff,
            LIM => pidLimited
        );

        // 3) Select output according to mode
        IF autoMode THEN
            controlOutputPct := yPID;
        ELSE
            controlOutputPct := manualCmd;
        END_IF

        // Clamp again for safety (Reforço dos limites)
        IF controlOutputPct < outLowLimitPct THEN controlOutputPct := outLowLimitPct; END_IF;
        IF controlOutputPct > outHighLimitPct THEN controlOutputPct := outHighLimitPct; END_IF;

        // 4) Exit to Idle when start is released or stop asserted
        IF NOT startCommand OR stopCommand THEN
            step := 90; // go to stopping
        END_IF

    // ------------------------------------------------------------
    90: // Stopping (Parando)
        controlOutputPct := 0.0;
        running := FALSE;
        step := 0;

    // ------------------------------------------------------------
    ELSE
        running := FALSE;
        controlOutputPct := 0.0;
        step := 0;
END_CASE

METHOD _InputFilter
VAR_INPUT
    enableFilter   : BOOL;  // TRUE=apply PT1, FALSE=bypass (TRUE=aplica PT1, FALSE=by-pass)
    rawValue       : REAL;  // Input value to be filtered (Valor de entrada a filtrar)
    filterTime     : TIME;  // PT1 time constant (Constante de tempo do PT1)
    filterGainK    : REAL;  // PT1 gain, typically 1.0 (Ganho do PT1, tipicamente 1.0)
END_VAR
VAR_OUTPUT
    filteredValue  : REAL;  // Filtered (or bypassed) value (Valor filtrado ou by-pass)
END_VAR
VAR
    kUse           : REAL;
    tUse           : TIME;
    yPT1           : REAL;
END_VAR
// When filter is disabled, "preload" the PT1 TO track the input quickly,
// so re-enabling is bumpless (sem degrau).
IF enableFilter THEN
    kUse := filterGainK;
    tUse := filterTime;
ELSE
    kUse := 1.0;          // track input
    tUse := T#10ms;       // tiny time constant
END_IF;

// Call the OSCAT PT1 filter instance
instsFT_PT1TInputFilter(
    in  := rawValue,
    T   := tUse,
    K   := kUse,
    out => yPT1
);

// Output selection
IF enableFilter THEN
    filteredValue := yPT1;
ELSE
    filteredValue := rawValue;
END_IF;
END_METHOD

END_FUNCTION_BLOCK

// ---- Function Blocks/PaperMachine/Auxiliary/FB_HeadboxLipsPWMControl.TcPOU
(*
    FB_HeadboxLipsPWMControl
    Purpose:
      - Control headbox lips opening using ON/OFF modulation (PWM), no analog speed output.
      - Manual: open/close while buttons are pressed (jog).
      - Automatic: operator types a target opening [mm] and presses "adjust"; the FB drives
        the lips toward the target using PWM duty proportional to position error magnitude.
      - If manualOpenCmd or manualCloseCmd is pressed during automatic positioning, the FB
        immediately returns to manual mode.

    Features:
      - Position units in millimeters (mm).
      - Limit sensors (limitMaxSensor / limitMinSensor) inhibit motion.
      - PWM duty [%] from |positionError| with clamps (min/max duty).
      - Minimum ON time per direction (minOnTime) to protect contactors.
      - Stall detection and travel timeout.
      - Exclusive actuation (never open & close simultaneously).
      - Human-readable deviceState.

    Notes:
      - Single PWM generator; direction is applied by gating its pulse.
      - Target is clamped to [posMin_mm .. posMax_mm].
*)

FUNCTION_BLOCK FB_HeadboxLipsPWMControl
VAR_INPUT
    // Position feedback and limits (mm)
    positionFeedback_mm     : REAL;          // Actual opening [mm]
    posMin_mm               : REAL := 0.0;   // Minimum allowed opening [mm]
    posMax_mm               : REAL := 25.0;  // Maximum allowed opening [mm]

    // Limit sensors
    limitMaxSensor          : BOOL;          // TRUE when fully open (max) limit is active
    limitMinSensor          : BOOL;          // TRUE when fully closed (min) limit is active

    // Manual jog commands (assume manual operation)
    manualOpenCmd           : BOOL;          // Jog open while pressed
    manualCloseCmd          : BOOL;          // Jog close while pressed

    // Automatic setpoint entry (assume automatic operation when pressed)
    autoTargetInput_mm      : REAL;          // Operator desired opening [mm]
    autoAdjustCmd           : BOOL;          // Pulse to start automatic positioning

    // Positioning behavior
    tolerance_mm            : REAL := 0.10;  // Position tolerance to finish [mm]

    // PWM behavior (OSCAT PWM_DC)
    pwmPeriod               : TIME := T#500ms; // PWM period
    pwmGainPct_per_mm       : REAL := 10.0;    // Duty slope: [% duty] per mm error
    pwmMinDutyPct           : REAL := 10.0;    // Minimum duty when moving [%]
    pwmMaxDutyPct           : REAL := 100.0;   // Maximum duty [%]

    // Contactor-friendly pulse shaping
    minOnTime               : TIME := T#300ms; // Minimum ON time per pulse/direction

    // Fault supervision
    stallDeltaMin_mm        : REAL := 0.02;    // Minimum position change to consider progress [mm]
    stallTimeout            : TIME := T#5s;    // No-progress duration => stall fault
    travelTimeout           : TIME := T#30s;   // Max time allowed to reach target => timeout fault
END_VAR

VAR_OUTPUT
    // Drive outputs (modulated by PWM in automatic mode)
    openingCmd              : BOOL;          // Command: open direction (PWM-modulated in Auto)
    closingCmd              : BOOL;          // Command: close direction (PWM-modulated in Auto)

    // Status
    busy                    : BOOL;          // TRUE while moving (Auto or Manual jog)
    done                    : BOOL;          // TRUE after successful auto positioning
    faultActive             : BOOL;          // Latched fault
    deviceState             : STRING(80);    // Human-readable state

    // Diagnostics
    target_mm               : REAL;          // Current target used [mm]
    positionError_mm        : REAL;          // Target - Feedback [mm]
    position_mm     : REAL;          			// Actual position [mm]	
    pwmDutyPct              : REAL;          // Current PWM duty commanded [%]
END_VAR

VAR
    // Mode / edges
    autoActive              : BOOL;          // Latched automatic mode (set by autoAdjustCmd, dropped by manual)
    autoAdjustOld           : BOOL;
    rAutoAdjust             : BOOL;

    // State machine
    step                    : INT;           // 0=Idle, 10=ManualOpen, 11=ManualClose, 20=AutoRun

    // Supervision
    lastPos_mm              : REAL;
    tonStall                : TON;
    tonTravel               : TON;

    // Helpers
    desiredTarget_mm        : REAL;          // Latched target on autoAdjust
    pwmPulse                : BOOL;          // PWM gate from OSCAT
    pwmEnable               : BOOL;          // Enable to PWM block
    needOpen                : BOOL;          // Direction: open (error > 0)
    needClose               : BOOL;          // Direction: close (error < 0)
    openPulseAllowed        : BOOL;          // PWM pulse after max limit check
    closePulseAllowed       : BOOL;          // PWM pulse after min limit check

    // Min-ON time timers per direction
    tonMinOnOpen            : TON;
    tonMinOnClose           : TON;

    // OSCAT instance
    instPWM                 : CTRL_PWM;        // Duty-cycle PWM generator (period-based)
END_VAR

// ============================== MAIN EXECUTION ==============================
rAutoAdjust := autoAdjustCmd AND NOT autoAdjustOld;
autoAdjustOld := autoAdjustCmd;

// Manual commands override automatic mode immediately
IF manualOpenCmd OR manualCloseCmd THEN
    autoActive := FALSE;            // leave automatic if any manual is pressed
END_IF;

// Latch automatic mode on adjust press
IF rAutoAdjust THEN
    autoActive := TRUE;
END_IF;

// Clear "done" on new auto adjust
IF rAutoAdjust THEN
    done := FALSE;
END_IF;

// Clear fault when fully idle (no manual pressed and not in auto)
IF (NOT manualOpenCmd) AND (NOT manualCloseCmd) AND (NOT autoActive) THEN
    faultActive := FALSE;
END_IF;

// Defaults
deviceState := 'Idle';
positionError_mm := target_mm - positionFeedback_mm;

// Abort on fault: de-energize outputs and stay idle
IF faultActive THEN
    _DriveNone();
    busy := FALSE;
    deviceState := 'Fault active';
    tonStall(IN:=FALSE);
    tonTravel(IN:=FALSE);
    tonMinOnOpen(IN:=FALSE);
    tonMinOnClose(IN:=FALSE);
ELSE
    // ========================== MANUAL OPERATION ==========================
    IF (manualOpenCmd XOR manualCloseCmd) AND (NOT autoActive) THEN
        // Only one manual command pressed => jog
        busy := TRUE;

		IF manualOpenCmd THEN
			IF limitMaxSensor OR (positionFeedback_mm >= posMax_mm) THEN
				_DriveNone();
				deviceState := 'Manual opening blocked: max limit (sensor/pos)';
			ELSE
				openingCmd := TRUE;
				closingCmd := FALSE;
				deviceState := 'Manual opening (jog)';
			END_IF
		
		ELSIF manualCloseCmd THEN
			IF limitMinSensor OR (positionFeedback_mm <= posMin_mm) THEN
				_DriveNone();
				deviceState := 'Manual closing blocked: min limit (sensor/pos)';
			ELSE
				closingCmd := TRUE;
				openingCmd := FALSE;
				deviceState := 'Manual closing (jog)';
			END_IF
		END_IF

        // Stop supervision in manual
        tonStall(IN:=FALSE);
        tonTravel(IN:=FALSE);
        tonMinOnOpen(IN:=FALSE);
        tonMinOnClose(IN:=FALSE);
        pwmDutyPct := 100.0; // purely diagnostic in manual jog

    ELSIF manualOpenCmd AND manualCloseCmd AND (NOT autoActive) THEN
        // Both pressed: conflict => stop
        busy := FALSE;
        _DriveNone();
        deviceState := 'Manual conflict (both pressed)';

        tonStall(IN:=FALSE);
        tonTravel(IN:=FALSE);
        tonMinOnOpen(IN:=FALSE);
        tonMinOnClose(IN:=FALSE);
        pwmDutyPct := 0.0;

    // ========================== AUTOMATIC OPERATION =======================
    ELSIF autoActive THEN
        // Latch target on rising edge of autoAdjust
        IF rAutoAdjust THEN
            desiredTarget_mm := _ClampReal(autoTargetInput_mm, posMin_mm, posMax_mm);
            target_mm := desiredTarget_mm;
            tonTravel(IN:=TRUE, PT:=travelTimeout);  // start travel timeout
            tonStall(IN:=FALSE);                     // arm stall after first measurement
            lastPos_mm := positionFeedback_mm;
        END_IF

        busy := TRUE;

        // Finish if within tolerance (no PWM pulses)
        IF _InTolerance(positionFeedback_mm, target_mm, tolerance_mm) THEN
            _DriveNone();
            busy := FALSE;
            done := TRUE;
            autoActive := FALSE; // auto move finished
            deviceState := 'Auto: in position';
            pwmDutyPct := 0.0;
            tonTravel(IN:=FALSE);
            tonStall(IN:=FALSE);
            tonMinOnOpen(IN:=FALSE);
            tonMinOnClose(IN:=FALSE);

        ELSE
            // Direction logic from error sign
            positionError_mm := target_mm - positionFeedback_mm;
            needOpen  := (positionError_mm > 0.0);
            needClose := (positionError_mm < 0.0);

            // Compute duty from error magnitude and clamp
            pwmDutyPct := _ErrorToDuty(ABS(positionError_mm), pwmGainPct_per_mm, pwmMinDutyPct, pwmMaxDutyPct);

            // Update PWM block (single generator, direction gating)
            pwmEnable := TRUE;
            _PwmUpdate(enable := pwmEnable, period := pwmPeriod, dutyPct := pwmDutyPct, pulse => pwmPulse);

            // Gate by limit sensors
            openPulseAllowed  := (needOpen  AND (NOT limitMaxSensor))  AND pwmPulse;
            closePulseAllowed := (needClose AND (NOT limitMinSensor)) AND pwmPulse;

            // Apply min-ON-time gating with exclusivity
            _ApplyMinOnGate(
                openPulseAllowed  := openPulseAllowed,
                closePulseAllowed := closePulseAllowed,
                minOnTime         := minOnTime,
                openingCmd        => openingCmd,
                closingCmd        => closingCmd
            );

            // Device state messages
            IF needOpen AND limitMaxSensor THEN
                deviceState := 'Auto opening blocked: max limit active';
            ELSIF needClose AND limitMinSensor THEN
                deviceState := 'Auto closing blocked: min limit active';
            ELSE
                IF needOpen THEN
                    deviceState := CONCAT('Auto opening (PWM ', REAL_TO_STRING(pwmDutyPct));
                ELSE
                    deviceState := CONCAT('Auto closing (PWM ', REAL_TO_STRING(pwmDutyPct));
                END_IF
            END_IF

            // Travel timeout supervision
            tonTravel(IN:=TRUE);

            // Stall detection: run timer when movement is too small
            IF ABS(positionFeedback_mm - lastPos_mm) < stallDeltaMin_mm THEN
                tonStall(IN:=TRUE, PT:=stallTimeout);
            ELSE
                tonStall(IN:=FALSE);
                lastPos_mm := positionFeedback_mm;
            END_IF

            // Faults
            IF tonTravel.Q THEN
                faultActive := TRUE;
                deviceState := 'Fault: travel timeout';
                _DriveNone();
                busy := FALSE;
                autoActive := FALSE;
                tonStall(IN:=FALSE);
                tonTravel(IN:=FALSE);
                tonMinOnOpen(IN:=FALSE);
                tonMinOnClose(IN:=FALSE);

            ELSIF tonStall.Q THEN
                faultActive := TRUE;
                deviceState := 'Fault: stall (no movement)';
                _DriveNone();
                busy := FALSE;
                autoActive := FALSE;
                tonStall(IN:=FALSE);
                tonTravel(IN:=FALSE);
                tonMinOnOpen(IN:=FALSE);
                tonMinOnClose(IN:=FALSE);
            END_IF
        END_IF

    // ========================== IDLE (no commands) ========================
    ELSE
        busy := FALSE;
        _DriveNone();
        deviceState := 'Idle';
        tonStall(IN:=FALSE);
        tonTravel(IN:=FALSE);
        tonMinOnOpen(IN:=FALSE);
        tonMinOnClose(IN:=FALSE);
        pwmDutyPct := 0.0;
    END_IF
END_IF


position_mm := positionFeedback_mm;

// ============================================================================
// METHOD: _ApplyMinOnGate
// Enforces a minimum ON-time for each direction and ensures exclusivity.
// - openPulseAllowed / closePulseAllowed are the post-limit PWM pulses.
// - Once a direction output turns ON, it stays ON for at least minOnTime.
// - While one direction is ON and still within its min ON-time, the other
//   direction cannot start (exclusivity).
// ============================================================================
METHOD PRIVATE _ApplyMinOnGate
VAR_INPUT
    openPulseAllowed   : BOOL;   // PWM pulse for OPEN, after limit check
    closePulseAllowed  : BOOL;   // PWM pulse for CLOSE, after limit check
    minOnTime          : TIME;   // Minimum ON time
END_VAR
VAR_OUTPUT
    openingCmd         : BOOL;   // Resulting OPEN command (after gating)
    closingCmd         : BOOL;   // Resulting CLOSE command (after gating)
END_VAR
// ---- OPEN direction gating ----
IF NOT openingCmd THEN
    // Eligible to start OPEN only if allowed pulse and CLOSE is not currently ON
    IF openPulseAllowed AND (NOT closingCmd) THEN
        openingCmd := TRUE;
        tonMinOnOpen(IN := TRUE, PT := minOnTime);
    ELSE
        openingCmd := FALSE;
        tonMinOnOpen(IN := FALSE);
    END_IF
ELSE
    // Currently ON: hold until min-ON elapsed; then follow pulse
    IF (NOT openPulseAllowed) AND tonMinOnOpen.Q THEN
        openingCmd := FALSE;
        tonMinOnOpen(IN := FALSE);
    ELSE
        // keep ON (either still within min-ON or pulse still present)
        tonMinOnOpen(IN := TRUE); // keep running; PT is ignored while already TRUE
    END_IF
END_IF

// Ensure exclusivity: if OPEN active, CLOSE must be off
IF openingCmd THEN
    closingCmd := FALSE;
    tonMinOnClose(IN := FALSE);
ELSE
    // ---- CLOSE direction gating (only if OPEN is not active) ----
    IF NOT closingCmd THEN
        IF closePulseAllowed AND (NOT openingCmd) THEN
            closingCmd := TRUE;
            tonMinOnClose(IN := TRUE, PT := minOnTime);
        ELSE
            closingCmd := FALSE;
            tonMinOnClose(IN := FALSE);
        END_IF
    ELSE
        IF (NOT closePulseAllowed) AND tonMinOnClose.Q THEN
            closingCmd := FALSE;
            tonMinOnClose(IN := FALSE);
        ELSE
            tonMinOnClose(IN := TRUE);
        END_IF
    END_IF
END_IF
END_METHOD

// ============================================================================
// METHOD: _ClampReal
// Returns val clamped to [lo..hi].
// ============================================================================
METHOD PRIVATE _ClampReal : REAL
VAR_INPUT
    val : REAL;
    lo  : REAL;
    hi  : REAL;
END_VAR
VAR
    v : REAL;
END_VAR


v := val;
IF v < lo THEN v := lo; END_IF;
IF v > hi THEN v := hi; END_IF;
_ClampReal := v;
END_METHOD

// ============================================================================
// METHOD: _DriveNone
// De-energize both outputs (exclusive safety).
// ============================================================================
METHOD PRIVATE _DriveNone
VAR_INPUT
END_VAR

openingCmd := FALSE;
closingCmd := FALSE;
END_METHOD

// ============================================================================
// METHOD: _ErrorToDuty
// Maps absolute error [mm] to PWM duty [%], with min/max clamps.
// duty = clamp( gain[%/mm] * absError_mm, minDuty%, maxDuty% )
// ============================================================================
METHOD PRIVATE _ErrorToDuty : REAL
VAR_INPUT
    absError_mm  : REAL;   // absolute position error [mm]
    gainPctPerMm : REAL;   // slope [% per mm]
    minDutyPct   : REAL;   // minimum duty [%]
    maxDutyPct   : REAL;   // maximum duty [%]
END_VAR
VAR
    d : REAL;
END_VAR


d := gainPctPerMm * absError_mm;
IF d < minDutyPct THEN d := minDutyPct; END_IF;
IF d > maxDutyPct THEN d := maxDutyPct; END_IF;
_ErrorToDuty := d;
END_METHOD



// ============================================================================
// METHOD: _InTolerance
// Returns TRUE when |value - target| <= tol
// ============================================================================
METHOD PRIVATE _InTolerance : BOOL
VAR_INPUT
    value   : REAL;
    target  : REAL;
    tol     : REAL;
END_VAR

_InTolerance := (ABS(value - target) <= tol);
END_METHOD

// ============================================================================
// METHOD: _PwmUpdate
// Updates OSCAT PWM_DC with enable, period and duty[%]. Returns pulse.
// NOTE: Adjust parameter names/types below if your OSCAT 'PWM_DC' signature differs.
// Common forms are: PWM_DC(EN, DC[% or 0..1], T, OUT) or (IN, DC, T, Q).
// ============================================================================
METHOD PRIVATE _PwmUpdate
VAR_INPUT
    enable   : BOOL;   // TRUE: PWM active, FALSE: output low
    period   : TIME;   // PWM period
    dutyPct  : REAL;   // Duty [%], 0..100
END_VAR
VAR_OUTPUT
    pulse    : BOOL;   // PWM output (TRUE during ON time)
END_VAR
VAR
    dcUse : REAL;
END_VAR


// Bound duty into 0..100%
dcUse := dutyPct;
IF dcUse < 0.0 THEN dcUse := 0.0; END_IF;
IF dcUse > 100.0 THEN dcUse := 100.0; END_IF;

// Call OSCAT PWM_DC
// If your PWM_DC expects 0..1 duty, divide by 100.0 here.
//instPWM(
//    EN := enable,          // enable
//    DC := dcUse,          // duty in percent (change to dcUse/100.0 if library expects 0..1)
//    T  := period,          // period
//    Q=> pulse            // boolean PWM output
//);

instPWM(
	CI:= dcUse * 0.01, 
	F:= 0.5, 
	Q=> pulse);
END_METHOD

END_FUNCTION_BLOCK

// ---- Function Blocks/PaperMachine/Auxiliary/FB_FormingBoardWireStretchControl.TcPOU
FUNCTION_BLOCK FB_FormingBoardWireStretchControl
VAR_INPUT
    stretchCmd           : BOOL;   // Jog command to stretch (increase tension)
    unstretchCmd         : BOOL;   // Jog command to unstretch (decrease tension)
    limitStretchSensor   : BOOL;   // TRUE when at maximum stretch limit
    limitUnstretchSensor : BOOL;   // TRUE when at minimum stretch limit
    fault                : BOOL;   // External fault interlock
END_VAR
VAR_OUTPUT
    stretch     : BOOL;           // Motor output: stretch direction
    unstretch   : BOOL;           // Motor output: unstretch direction
    busy        : BOOL;           // TRUE when motor running in any direction
    deviceState : STRING(80);     // Human-readable status for HMI
END_VAR

// ============================ MAIN EXECUTION ============================

// Safety: External fault forces outputs OFF
IF fault THEN
    stretch := FALSE;
    unstretch := FALSE;
    busy := FALSE;
    deviceState := 'Fault active';

ELSE
    // Conflict handling: both commands pressed
    IF stretchCmd AND unstretchCmd THEN
        stretch := FALSE;
        unstretch := FALSE;
        busy := FALSE;
        deviceState := 'Conflict: both commands pressed';

    ELSE
        // ======================= STRETCH control ========================
        IF stretchCmd AND NOT limitStretchSensor AND NOT unstretchCmd THEN
            stretch := TRUE;
        ELSE
            stretch := FALSE;
        END_IF

        // ======================= UNSTRETCH control ======================
        IF unstretchCmd AND NOT limitUnstretchSensor AND NOT stretchCmd THEN
            unstretch := TRUE;
        ELSE
            unstretch := FALSE;
        END_IF

        // ======================= State / Busy flag ======================
        busy := stretch OR unstretch;

        IF stretch THEN
            IF limitStretchSensor THEN
                deviceState := 'Stretch blocked: max limit';
            ELSE
                deviceState := 'Stretching...';
            END_IF
        ELSIF unstretch THEN
            IF limitUnstretchSensor THEN
                deviceState := 'Unstretch blocked: min limit';
            ELSE
                deviceState := 'Unstretching...';
            END_IF
        ELSE
            deviceState := 'Idle';
        END_IF
    END_IF
END_IF

END_FUNCTION_BLOCK

// ---- Function Blocks/PaperMachine/Auxiliary/FB_LevelControl_V2.TcPOU
(*
  Change summary (minimal):
    - Added reverseActing : BOOL := TRUE  // default for draining pumps
    - Added kpUse : REAL
    - PID now uses KP := kpUse where kpUse = ±ABS(kp) depending on reverseActing
*)

FUNCTION_BLOCK FB_LevelControl_V2
VAR_INPUT
    // ===== Sequence commands =====
    startCommand            : BOOL;            // Start pulse (toggle run)
    stopCommand             : BOOL;            // Stop pulse/level (force stop)

    // ===== Mode =====
    autoMode                : BOOL;            // TRUE=Automatic / FALSE=Manual

    // ===== Process signals (LEVEL) =====
    levelFeedbackEng        : REAL;            // Level feedback (engineering units)
    levelSetpointEng        : REAL;            // Setpoint in engineering units

    // ===== Manual output (direct % to final element) =====
    manualOutputPct         : REAL;            // 0..100% manual output

    // ===== PID parameters (OSCAT CTRL_PID) =====
    kp                      : REAL := 1.0;     // proportional gain (magnitude; sign handled by reverseActing)
    tn                      : REAL := 8.0;     // integral time [s]
    tv                      : REAL := 0.0;     // derivative time [s]
    deadBand				: REAL := 0.0;     // PID DeadBand
	
    // ===== NEW: Reverse/Direct action selector =====
    reverseActing           : BOOL := TRUE;    // TRUE = reverse action (draining pump default)

    // ===== Output limits & offset =====
    outLowLimitPct          : REAL := 0.0;
    outHighLimitPct         : REAL := 100.0;
    outputOffsetPct         : REAL := 0.0;     // added to final output

    // ===== PID housekeeping =====
    resetPID                : BOOL;            // reset integrator

    // ===== Input filter (OSCAT PT1) =====
    enableInputFilter       : BOOL := TRUE;
    inputFilterTime         : TIME := T#500ms;
    inputFilterGainK        : REAL := 1.0;
	
    displayFilterTime       : TIME := T#20MS;	
	

    // ===== Optional scaling (engineering <-> %) =====
    enableScaling           : BOOL := TRUE;
    lvlLoEng                : REAL := 0.0;
    lvlHiEng                : REAL := 100.0;

    // ===== VFD interface & supervision =====
    vfdReady                : BOOL;            // VFD ready/healthy
    vfdRunFeedback          : BOOL;            // VFD RUN feedback
    vfdFaultFeedback        : BOOL;            // VFD fault feedback
    vfdRunFbTimeout         : TIME := T#5s;    // Timeout to receive RUN FB after start

    // ===== VFD analog feedbacks =====
    vfdCurrentFeedback      : REAL;            // Motor current [A]
    vfdEngFeedback          : REAL;            // Motor enginering feedback
    vfdTorqueFeedback       : REAL;            // Motor torque feedback
	

    // ===== SAFETY (true safety only) =====
    safetyOk                : BOOL := TRUE;    // Safety relay / chain OK
    estopOk                 : BOOL := TRUE;    // E-Stop loop OK
    guardClosedOk           : BOOL := TRUE;    // Doors/guards closed

    // ===== INTERLOCKS (process permissives) — NORMAL STOP ONLY =====
    interlock1              : BOOL := TRUE;
    interlock2              : BOOL := TRUE;
    interlock3              : BOOL := TRUE;
    interlock4              : BOOL := TRUE;
    interlock5              : BOOL := TRUE;
    interlock6              : BOOL := TRUE;

    // ===== Minimum level supervision (process permissive) =====
    minLevelEnable          : BOOL := TRUE;    // Enable low-level stop/hold logic
    minLevelStopEng         : REAL := 10.0;    // Trip threshold (Eng units) => stop & hold
    minLevelRestartEng      : REAL := 12.0;    // Release threshold (Eng units) => auto restart
    minLevelTripTime        : TIME := T#1s;    // Level < StopEng for this long to trip
    minLevelReleaseTime     : TIME := T#1s;    // Level > RestartEng for this long to release
END_VAR

VAR_OUTPUT
    running                 : BOOL;            // TRUE only in RUN (use to release other devices)
    controlOutputPct        : REAL;            // 0..100 %
    pidDiff                 : REAL;            // SET - ACT (post-scaling)
    pidLimited              : BOOL;            // TRUE if saturated
    deviceState             : STRING(80);      // Human-readable state
    vfdStartCmdOut          : BOOL;            // Asserted in Starting/Running (VFD START)
    minLevelHoldActive      : BOOL;            // TRUE while in low-level hold

    // Status & displays
    statusCode              : INT;             // 0=Idle, 1=Running, 2=Fault
    vfdCurrentDisplay       : REAL;            // Displayed motor current [A]
    vfdTorqueDisplay       : REAL;            // Displayed motor current [A]
    vfdEngDisplay           : REAL;            // Displayed motor speed [rpm]
	levelDisplay			: REAL;
	
END_VAR

VAR
    // ===== State & edges =====
    step                    : INT;             // 0=Idle,10=Starting,20=Running,90=Stopping
    startOld                : BOOL;
    stopOld                 : BOOL;
    rStart                  : BOOL;            // start pulse edge
    rStop                   : BOOL;            // stop pulse edge
    runLatch                : BOOL;            // toggled by Start; cleared by Stop

    // ===== Internals =====
    manualCmd               : REAL;
    yPID                    : REAL;
    kpUse                   : REAL;            // sign-adjusted Kp

    // Filtered PV (engineering)
    levelFeedbackEngFilt    : REAL;

    // PV/SP in %
    pvPct                   : REAL;
    spPct                   : REAL;

    // Timers / supervision
    tonRunFbWait            : TON;

    // Minimum level timers/flags
    minLevelBelow           : BOOL;
    minLevelAboveRestart    : BOOL;
    tonMinLevelTrip         : TON;
    tonMinLevelRelease      : TON;

    // Instances
    instPID                 : CTRL_PID;
    instPT1                 : FT_PT1;

    // Aggregations
    allSafetyOK             : BOOL;
    anyInterlockOpen        : BOOL;
	
    instPT1_TorqueDisplay  		: FT_PT1;
    instPT1_SpeedDisplay   		: FT_PT1;
    instPT1_LevelDisplay   		: FT_PT1;

	
END_VAR

// ============================ Edges ============================
rStart := startCommand AND NOT startOld;
startOld := startCommand;

rStop  := stopCommand AND NOT stopOld;
stopOld := stopCommand;

// Start toggles run; Stop forces stop
IF rStart THEN
    runLatch := NOT runLatch;
END_IF;
IF rStop OR stopCommand THEN
    runLatch := FALSE;
END_IF;


// ============================ Aggregations =====================
allSafetyOK := safetyOk AND estopOk AND guardClosedOk;
anyInterlockOpen := NOT (interlock1 AND interlock2 AND interlock3 AND interlock4 AND interlock5 AND interlock6);

// Defaults each cycle
vfdStartCmdOut := FALSE;




// ============================ Minimum level supervision ============================
// Compare using current engineering PV (raw). If preferred, swap to levelFeedbackEngFilt.
minLevelBelow        := (levelFeedbackEng <  minLevelStopEng);
minLevelAboveRestart := (levelFeedbackEng >  minLevelRestartEng);

IF minLevelEnable THEN
    // Trip debounce
    tonMinLevelTrip(IN := minLevelBelow, PT := minLevelTripTime);
    // Release debounce
    tonMinLevelRelease(IN := minLevelAboveRestart, PT := minLevelReleaseTime);

    // Latch HOLD on trip, clear on release
    IF tonMinLevelTrip.Q THEN
        minLevelHoldActive := TRUE;
    END_IF;
    IF tonMinLevelRelease.Q THEN
        minLevelHoldActive := FALSE;
    END_IF;
ELSE
    tonMinLevelTrip(IN := FALSE);
    tonMinLevelRelease(IN := FALSE);
    minLevelHoldActive := FALSE;
END_IF;


// ============================ Immediate stop / safety/fault guards ============
IF rStop OR stopCommand THEN
    controlOutputPct := 0.0;
    running := FALSE;
    deviceState := 'Stopping (Stop command)';
    runLatch := FALSE;                    // ensure toggled off
    step := 90;
END_IF;

IF vfdFaultFeedback THEN
    deviceState := 'Fault from VFD';
    runLatch := FALSE;
    step := 90;
END_IF;

IF NOT allSafetyOK THEN
    deviceState := 'Stopping: Safety chain open';
    runLatch := FALSE;
    step := 90;
END_IF;


// ============================ State machine =====================
CASE step OF
    // ------------------------------------------------------------
    0: // Idle
        running := FALSE;
        controlOutputPct := 0.0;
        deviceState := 'Idle';
        vfdStartCmdOut := FALSE;

        // Start request via runLatch (toggled by Start pulse)
        IF runLatch AND NOT stopCommand THEN
            // Safety must be OK; VFD must be ready; min level must not be holding
            IF NOT allSafetyOK THEN
                deviceState := 'Start blocked: Safety not OK';
                runLatch := FALSE; // block and clear latch to avoid re-trigger
                step := 0;
            ELSIF NOT vfdReady THEN
                deviceState := 'Start blocked: VFD not ready';
                runLatch := FALSE;
                step := 0;
            ELSIF minLevelEnable AND minLevelHoldActive THEN
                deviceState := 'Start blocked: Low level hold';
                runLatch := FALSE;
                step := 0;
            ELSE
                deviceState := 'Starting';
                vfdStartCmdOut := TRUE;                   // send START to VFD
                tonRunFbWait(IN := TRUE, PT := vfdRunFbTimeout);
                step := 10;
            END_IF
        END_IF

    // ------------------------------------------------------------
    10: // Starting (await RUN feedback)
        running := FALSE;
        deviceState := 'Starting (await RUN fb)';
        vfdStartCmdOut := TRUE;

        // Safety/fault during start => stop
        IF NOT allSafetyOK THEN
            tonRunFbWait(IN := FALSE);
            deviceState := 'Stopping: Safety chain open';
            vfdStartCmdOut := FALSE;
            runLatch := FALSE;
            step := 90;

        ELSIF vfdFaultFeedback THEN
            tonRunFbWait(IN := FALSE);
            deviceState := 'Fault from VFD';
            vfdStartCmdOut := FALSE;
            runLatch := FALSE;
            step := 90;

        // Interlocks are normal stop only
        ELSIF anyInterlockOpen THEN
            tonRunFbWait(IN := FALSE);
            deviceState := 'Stopping: Interlock open';
            vfdStartCmdOut := FALSE;
            runLatch := FALSE;
            step := 90;

        // Minimum level HOLD => normal stop
        ELSIF minLevelEnable AND minLevelHoldActive THEN
            tonRunFbWait(IN := FALSE);
            deviceState := 'Stopping: Low level hold';
            vfdStartCmdOut := FALSE;
            runLatch := FALSE;
            step := 90;

        // RUN fb arrived
        ELSIF vfdRunFeedback THEN
            tonRunFbWait(IN := FALSE);
            step := 20;

        // Timeout
        ELSIF tonRunFbWait.Q THEN
            tonRunFbWait(IN := FALSE);
            deviceState := 'Start failed: RUN feedback timeout';
            vfdStartCmdOut := FALSE;
            runLatch := FALSE;
            step := 90;
        END_IF

    // ------------------------------------------------------------
    20: // Running (control loop)
        running := TRUE;               // release other devices with this
        deviceState := 'Running';
        vfdStartCmdOut := TRUE;

        // Supervision
        IF NOT allSafetyOK THEN
            deviceState := 'Stopping: Safety chain open';
            vfdStartCmdOut := FALSE;
            runLatch := FALSE;
            step := 90;

        ELSIF vfdFaultFeedback THEN
            deviceState := 'Fault from VFD';
            vfdStartCmdOut := FALSE;
            runLatch := FALSE;
            step := 90;

        ELSIF NOT vfdReady THEN
            deviceState := 'Stopping: VFD not ready';
            vfdStartCmdOut := FALSE;
            runLatch := FALSE;
            step := 90;

        ELSIF NOT vfdRunFeedback THEN
            deviceState := 'Stopping: RUN feedback lost';
            vfdStartCmdOut := FALSE;
            runLatch := FALSE;
            step := 90;

        // INTERLOCKS → NORMAL STOP ONLY
        ELSIF anyInterlockOpen THEN
            deviceState := 'Stopping: Interlock open';
            vfdStartCmdOut := FALSE;
            runLatch := FALSE;
            step := 90;

        // Minimum level HOLD → NORMAL STOP
        ELSIF minLevelEnable AND minLevelHoldActive THEN
            deviceState := 'Stopping: Low level hold';
            vfdStartCmdOut := FALSE;
            runLatch := FALSE;
            step := 90;

        // Start toggled OFF while running => stop
        ELSIF NOT runLatch THEN
            deviceState := 'Stopping (Start toggled off)';
            vfdStartCmdOut := FALSE;
            step := 90;

        ELSE
            // ---- Input filtering (PT1) ----
            IF enableInputFilter THEN
                instPT1(in := levelFeedbackEng, T := inputFilterTime, K := inputFilterGainK, out => levelFeedbackEngFilt);
            ELSE
                levelFeedbackEngFilt := levelFeedbackEng;
            END_IF

            // ---- Engineering -> % scaling ----
            IF enableScaling THEN
                pvPct := _ScaleToPct(levelFeedbackEngFilt, lvlLoEng, lvlHiEng);
                spPct := _ScaleToPct(levelSetpointEng,     lvlLoEng, lvlHiEng);
            ELSE
                pvPct := levelFeedbackEngFilt;    // already %
                spPct := levelSetpointEng;        // already %
            END_IF

            // ---- Manual path and PID with bumpless transfer ----
            manualCmd := LIMIT(0.0, manualOutputPct, 100.0);

            // Reverse/direct action by Kp sign
            IF reverseActing THEN
                kpUse := -ABS(kp);
            ELSE
                kpUse :=  ABS(kp);
            END_IF

            instPID(
                ACT := pvPct,
                SET := spPct,
                M_I := manualCmd,
                MAN := NOT autoMode,
                RST := resetPID,
                KP  := kpUse,              // <— inverted when reverseActing=TRUE
                TN  := tn,
                TV  := tv,
				SUP := deadBand,
                LL  := outLowLimitPct,
                LH  := outHighLimitPct,
                Y   => yPID,
                DIFF=> pidDiff,
                LIM => pidLimited
            );

            // Mode select, offset, clamp
            IF autoMode THEN
                controlOutputPct := yPID;
            ELSE
                controlOutputPct := manualCmd;
            END_IF
            controlOutputPct := LIMIT(outLowLimitPct, controlOutputPct + outputOffsetPct, outHighLimitPct);
        END_IF

    // ------------------------------------------------------------
    90: // Stopping (normal, de-energize)
        running := FALSE;
        controlOutputPct := 0.0;
        vfdStartCmdOut := FALSE;
        tonRunFbWait(IN := FALSE);

        // Return to Idle once stop released and safety OK
        IF NOT stopCommand AND allSafetyOK THEN
            deviceState := 'Idle';
            step := 0;
        END_IF

    // ------------------------------------------------------------
    ELSE
        running := FALSE;
        controlOutputPct := 0.0;
        deviceState := 'Idle';
        vfdStartCmdOut := FALSE;
        step := 0;
END_CASE


// =============================== Status code =======================================
IF vfdFaultFeedback THEN
    statusCode := 2;             // Fault
ELSIF running THEN
    statusCode := 1;             // Running
ELSE
    statusCode := 0;             // Idle
END_IF


_FeedbackDisplay();

METHOD _FeedbackDisplay
VAR_INPUT
END_VAR
// 5) HMI DISPLAY SIGNALS (filtered speeds/torques + GROUP status)
instPT1_SpeedDisplay(in := vfdEngFeedback, T := displayFilterTime, K := 1.0, out => vfdEngDisplay);
instPT1_TorqueDisplay (in := vfdTorqueFeedback , T := displayFilterTime, K := 1.0, out => vfdTorqueDisplay);
instPT1_LevelDisplay (in := levelFeedbackEng , T := displayFilterTime, K := 1.0, out => levelDisplay);
END_METHOD

// ============================ Helper ============================
METHOD PRIVATE _ScaleToPct : REAL
VAR_INPUT
    xEng  : REAL;  // value in engineering units
    loEng : REAL;  // min eng
    hiEng : REAL;  // max eng
END_VAR
VAR
    span : REAL;
    pct  : REAL;
END_VAR

span := hiEng - loEng;
IF span = 0.0 THEN
    _ScaleToPct := 0.0; // avoid div by zero
ELSE
    pct := (xEng - loEng) / span * 100.0;
    _ScaleToPct := LIMIT(0.0, pct, 100.0);
END_IF
END_METHOD

END_FUNCTION_BLOCK

// ---- Function Blocks/PaperMachine/Auxiliary/FB_WirePitControl.TcPOU
(*
    FB_ProcessControler
    Purpose: Generic process controller with start/stop latch, status codes,
             PID (OSCAT CTRL_PID), optional reverse action, PV PT1 filter,
             engineering↔% scaling, drive run supervision, and HMI displays.

    Sequence: Start pulse toggles RUN latch; Stop pulse/level forces stop.

    Status codes: statusCode INT → 0=Idle, 1=Running, 2=Fault

    Notes: Includes optional low/high PV “hold” with hysteresis (normal-stop class).
*)

FUNCTION_BLOCK FB_WirePitControl
VAR_INPUT
    // ===== Sequence commands =====
    startCommand                 : BOOL;            // Start pulse toggles RUN latch
    stopCommand                  : BOOL;            // Stop pulse/level forces stop

    // ===== Manual output & Auto SP nudge =====
    processSetpointManInc        : BOOL;            // Manual output ↑ (0..100%)
    processSetpointManDec        : BOOL;            // Manual output ↓ (0..100%)
    processSetpointManSteps      : REAL := 0.1;

    processSetpointAutoInc       : BOOL;            // Auto SP ↑ (engineering units or %)
    processSetpointAutoDec       : BOOL;            // Auto SP ↓ (engineering units or %)
    processSetpointAutoSteps     : REAL := 1.0;

    // ===== Mode =====
    autoMode                     : BOOL;            // TRUE=Automatic / FALSE=Manual
    reverseActing                : BOOL := FALSE;   // TRUE: higher output decreases PV; FALSE: direct

    // ===== Process signals (PV in engineering units) =====
    wirePitLevel           : REAL;            // PV (engineering units), e.g., bar/kPa/°C/…
	whiteWaterSiloLevel			: REAL;
    // ===== PID parameters (OSCAT CTRL_PID) =====
    kp                           : REAL := 1.0;     // Proportional gain (sign handled via reverseActing)
    tn                           : REAL := 8.0;     // Integral time [s]
    tv                           : REAL := 0.0;     // Derivative time [s]

    // ===== Output limits & offset =====
    outLowLimitPct               : REAL := 0.0;     // Min output %
    outHighLimitPct              : REAL := 100.0;   // Max output %
    outputOffsetPct              : REAL := 0.0;     // Offset added to final output

    // ===== PID housekeeping =====
    resetPID                     : BOOL;            // Reset integrator

    // ===== Input filter (OSCAT FT_PT1) =====
    enableInputFilter            : BOOL := TRUE;    // Enable PV PT1 filter
    inputFilterTime              : TIME := T#300ms; // PT1 time constant
    inputFilterGainK             : REAL := 1.0;     // PT1 gain

    displayFilterTime            : TIME := T#20ms;  // Small PT1 for HMI displays

    // ===== Optional scaling (engineering ↔ %) =====
    enableScaling                : BOOL := TRUE;    // Enable engineering↔% scaling
    pLoEng                       : REAL := 0.0;     // Engineering low bound
    pHiEng                       : REAL := 10.0;    // Engineering high bound

    // ===== Drive interface & supervision (VFD or actuator drive) =====
    vfdReady                     : BOOL;            // Drive ready/healthy
    vfdRunFeedback               : BOOL;            // Drive RUN feedback
    vfdFaultFeedback             : BOOL;            // Drive fault
    vfdRunFbTimeout              : TIME := T#5s;    // Timeout to receive RUN FB after start

    // ===== Drive analog feedbacks (for HMI display) =====
    vfdCurrentFeedback           : REAL;            // Current [A or %]
    vfdEngFeedback               : REAL;            // Engineering feedback (e.g., rpm, flow, etc.)
    vfdTorqueFeedback            : REAL;            // Torque (Nm or %)

    // ===== Safety (true safety inputs only) =====
    safetyOk                     : BOOL := TRUE;    // Safety chain OK
    estopOk                      : BOOL := TRUE;    // E-Stop loop OK
    guardClosedOk                : BOOL := TRUE;    // Guards/doors closed

    // ===== Interlocks (process permissives) — normal stop only =====
    interlock1                   : BOOL := TRUE;
    interlock2                   : BOOL := TRUE;
    interlock3                   : BOOL := TRUE;
    interlock4                   : BOOL := TRUE;
    interlock5                   : BOOL := TRUE;
    interlock6                   : BOOL := TRUE;

 // ===== Optional low-PV hold (normal-stop/hold) =====
    minPVEnable                  : BOOL := FALSE;   // Enable low-PV hold
    minPVTripEng                 : REAL := 0.5;     // Trip threshold (engineering units)
    minPVReleaseEng              : REAL := 0.7;     // Release threshold (engineering units)
    minPVTripTime                : TIME := T#1s;    // PV < trip for this long to trip
    minPVReleaseTime             : TIME := T#1s;    // PV > release for this long to release

    // ===== Optional high-PV hold (normal-stop/hold) =====
    maxPVEnable                  : BOOL := FALSE;   // Enable high-PV hold
    maxPVTripEng                 : REAL := 9.5;     // Trip threshold (engineering units)
    maxPVReleaseEng              : REAL := 9.2;     // Release threshold (engineering units)
    maxPVTripTime                : TIME := T#1s;    // PV > trip for this long to trip
    maxPVReleaseTime             : TIME := T#1s;    // PV < release for this long to release
	
	
END_VAR

VAR_OUTPUT
    running                      : BOOL;            // TRUE only during RUN state
    controlOutputPct             : REAL;            // Final control output 0..100%
    pidDiff                      : REAL;            // SET − ACT (post-scaling)
    pidLimited                   : BOOL;            // TRUE if saturated
    deviceState                  : STRING(80);      // Human-readable state
    vfdStartCmdOut               : BOOL;            // Asserted in Start/Run to the drive

    // ===== Holds (normal stop class) =====
    minPressureHoldActive        : BOOL;            // Low-PV hold active
    maxPressureHoldActive        : BOOL;            // High-PV hold active

    // ===== Status & HMI displays =====
    statusCode                   : INT;             // 0=Idle, 1=Running, 2=Fault
    vfdCurrentDisplay            : REAL;            // Display current [A or %]
    vfdTorqueDisplay             : REAL;            // Display torque (Nm or %)
    vfdEngDisplay                : REAL;            // Display engineering feedback (e.g., rpm)
    wirePitLevelDisplay    : REAL;            // PV (engineering units), e.g., bar/kPa/°C/…
	whiteWaterSiloLevelDisplay		: REAL;
	
END_VAR

VAR
    // ===== First scan & state/edges =====
    firstScan                    : BOOL := TRUE;    // TRUE only on first PLC cycle
	pvHoldActive  				 : BOOL;  
    step                         : INT;             // 0=Idle,10=Starting,20=Running,90=Stopping
    startOld                     : BOOL;            // Edge memory
    stopOld                      : BOOL;            // Edge memory
    rStart                       : BOOL;            // Rising edge: start
    rStop                        : BOOL;            // Rising edge: stop
    runLatch                     : BOOL;            // Toggled by Start; cleared by Stop

    // ===== Internals =====
    manualCmd                    : REAL;            // Manual command %
    yPID                         : REAL;            // PID output %
    kpUse                        : REAL;            // Kp adjusted by reverseActing

    // ===== Filtered PV (engineering units) =====
    pvEngFiltered                : REAL;

    // ===== PV & SP in % (post-scaling) =====
    pvPct                        : REAL;
    spPct                        : REAL;

    // ===== Timers =====
    tonRunFbWait                 : TON;             // Waits RUN FB after start

    // ===== Low/High PV timers =====
    tonMinPTrip                  : TON;
    tonMinPRelease               : TON;
    tonMaxPTrip                  : TON;
    tonMaxPRelease               : TON;

    // ===== Instances =====
    instPID                      : CTRL_PID;        // OSCAT PID
    instPT1                      : FT_PT1;          // PV PT1 filter

    // ===== Aggregations =====
    allSafetyOK                  : BOOL;            // safetyOk & estopOk & guardClosedOk
    anyInterlockOpen             : BOOL;            // any interlock is FALSE

    // ===== HMI display filters =====
    instPT1_TorqueDisplay        : FT_PT1;          // PT1 for torque display
    instPT1_SpeedDisplay         : FT_PT1;          // PT1 for engineering display
	
    instPT1_ProcessFeedbackEngDisplay        : FT_PT1;          // PT1 for engineering display
	instPT1_WhiteWaterSiloLevelDisplay        : FT_PT1;          // PT1 for engineering display


    processSetpointManOld        : REAL;            // Last observed manual SP (HMI)
    processSetpointAutoOld       : REAL;            // Last observed auto SP (HMI)
	minPVHoldActive: BOOL;
	maxPVHoldActive: BOOL;
END_VAR

VAR PERSISTENT
    instTUNE2AutoSetpoint        : TUNE2;           // OSCAT TUNE2 for auto SP nudge
    instTUNE2ManSetpoint         : TUNE2;           // OSCAT TUNE2 for manual output
END_VAR

VAR_IN_OUT
    // ===== Exposed setpoints =====
    processSetpointMan           : REAL;            // Manual output 0..100%
    processSetpointAuto          : REAL;            // Auto SP (engineering units or % per configuration)
END_VAR

// ============================ INITIALIZATION ============================
// Run this block only once on first cycle
IF firstScan THEN
    firstScan := FALSE;

    processSetpointMan      := instTUNE2ManSetpoint.Y;
    processSetpointManOld   := processSetpointMan;

    processSetpointAuto     := instTUNE2AutoSetpoint.Y;
    processSetpointAutoOld  := processSetpointAuto;
END_IF;


// ============================ Edges ============================
rStart := startCommand AND NOT startOld;
startOld := startCommand;

rStop  := stopCommand AND NOT stopOld;
stopOld := stopCommand;

// Start toggles run; Stop forces stop
IF rStart THEN
    runLatch := TRUE;
END_IF;
IF rStop OR stopCommand THEN
    runLatch := FALSE;
END_IF;


// ============================ Aggregations =====================
allSafetyOK := safetyOk AND estopOk AND guardClosedOk;
anyInterlockOpen := NOT (interlock1 AND interlock2 AND interlock3 AND interlock4 AND interlock5 AND interlock6);

// Defaults each cycle
vfdStartCmdOut := FALSE;


// ============================ Low/High PV HOLD supervision ============================
// LOW-PV - Hold if the wire pit level is too low
IF minPVEnable AND autoMode THEN
    tonMinPTrip   (IN := (wirePitLevel <  minPVTripEng),     PT := minPVTripTime);
    tonMinPRelease(IN := (wirePitLevel >  minPVReleaseEng),  PT := minPVReleaseTime);
    IF tonMinPTrip.Q    THEN minPVHoldActive := TRUE;  END_IF;
    IF tonMinPRelease.Q THEN minPVHoldActive := FALSE; END_IF;

ELSE
    tonMinPTrip(IN := FALSE);
    tonMinPRelease(IN := FALSE);
    minPVHoldActive := FALSE;
END_IF;

